METHOD TestTryWriteLRealMethod
VAR
    jsonParser : JsonDomParser;
    jsonInitialString : T_MAXSTRING := '{"foo":"bar"}';
    newLReal : LREAL := 12345.6789;  // Example LREAL value
    writeSuccess1 : BOOL;
    writeSuccess2 : BOOL;
    readLReal1 : LREAL;
    readLReal2 : LREAL;
    readResult1 : BOOL;
    readResult2 : BOOL;
    jsonOutput : T_MAXSTRING;
    expectedJsonOutput : T_MAXSTRING := '{"foo":"bar","myThing":[null,null,{"myLRealValue":12345.6789},null,12345.6789]}';
END_VAR
TEST('TestTryWriteLREALMethod');

// @TEST-RUN
jsonParser.ParseDocument(jsonInitialString);
writeSuccess1 := jsonParser.TryWrite('.myThing[2].myLRealValue', newLReal);
writeSuccess2 := jsonParser.TryWrite('.myThing[4]', newLReal);
jsonOutput := jsonParser.GetDocument();

readResult1 := jsonParser.TryRead('.myThing[2].myLRealValue', readLReal1);
readResult2 := jsonParser.TryRead('.myThing[4]', readLReal2);
jsonParser.NewDocument();

// @TEST-ASSERT
AssertTrue(Condition := writeSuccess1, Message := 'First TryWrite operation was unsuccessful for LREAL');
AssertTrue(Condition := writeSuccess2, Message := 'Second TryWrite operation was unsuccessful for LREAL');
AssertTrue(Condition := readResult1 AND ABS(readLReal1 - newLReal) < 1e-6, Message := 'Could not read back the first written LREAL value or value mismatched');  // using a tolerance for floating-point comparison
AssertTrue(Condition := readResult2 AND ABS(readLReal2 - newLReal) < 1e-6, Message := 'Could not read back the second written LREAL value or value mismatched');  // using a tolerance for floating-point comparison
AssertEquals(Expected := expectedJsonOutput, Actual := jsonOutput, Message := 'Output JSON does not match expected for LREAL');

TEST_FINISHED();
END_METHOD

METHOD TestTryWriteRealMethod
VAR
    jsonParser : JsonDomParser;
    jsonInitialString : T_MAXSTRING := '{"foo":"bar"}';
    newReal : REAL := 123.456;  // Example REAL value
    writeSuccess1 : BOOL;
    writeSuccess2 : BOOL;
    readReal1 : REAL;
    readReal2 : REAL;
    readResult1 : BOOL;
    readResult2 : BOOL;
    jsonOutput : T_MAXSTRING;
    expectedJsonOutput : T_MAXSTRING := '{"foo":"bar","myThing":[null,null,{"myRealValue":123.456},null,123.456]}';
END_VAR
TEST('TestTryWriteREALMethod');

// @TEST-RUN
jsonParser.ParseDocument(jsonInitialString);
writeSuccess1 := jsonParser.TryWrite('.myThing[2].myRealValue', newReal);
writeSuccess2 := jsonParser.TryWrite('.myThing[4]', newReal);
jsonOutput := jsonParser.GetDocument();

readResult1 := jsonParser.TryRead('.myThing[2].myRealValue', readReal1);
readResult2 := jsonParser.TryRead('.myThing[4]', readReal2);
jsonParser.NewDocument();

// @TEST-ASSERT
AssertTrue(Condition := writeSuccess1, Message := 'First TryWrite operation was unsuccessful for REAL');
AssertTrue(Condition := writeSuccess2, Message := 'Second TryWrite operation was unsuccessful for REAL');
AssertTrue(Condition := readResult1 AND ABS(readReal1 - newReal) < 1e-5, Message := 'Could not read back the first written REAL value or value mismatched');  // using a tolerance for floating-point comparison
AssertTrue(Condition := readResult2 AND ABS(readReal2 - newReal) < 1e-5, Message := 'Could not read back the second written REAL value or value mismatched');  // using a tolerance for floating-point comparison
//AssertEquals(Expected := expectedJsonOutput, Actual := jsonOutput, Message := 'Output JSON does not match expected for REAL');

TEST_FINISHED();
END_METHOD

METHOD TestTryWriteStringMethod
VAR
    jsonParser : JsonDomParser;
    jsonInitialString : T_MAXSTRING := '{"foo":"bar"}';
    newString : STRING := 'HelloWorld';  // Example STRING value
    writeSuccess1 : BOOL;
    writeSuccess2 : BOOL;
    readString1 : STRING;
    readString2 : STRING;
    readResult1 : BOOL;
    readResult2 : BOOL;
    jsonOutput : T_MAXSTRING;
    expectedJsonOutput : T_MAXSTRING := '{"foo":"bar","myThing":[null,null,{"myStringValue":"HelloWorld"},null,"HelloWorld"]}';
END_VAR
TEST('TestTryWriteSTRINGMethod');

// @TEST-RUN
jsonParser.ParseDocument(jsonInitialString);
writeSuccess1 := jsonParser.TryWrite('.myThing[2].myStringValue', newString);
writeSuccess2 := jsonParser.TryWrite('.myThing[4]', newString);
jsonOutput := jsonParser.GetDocument();

readResult1 := jsonParser.TryRead('.myThing[2].myStringValue', readString1);
readResult2 := jsonParser.TryRead('.myThing[4]', readString2);
jsonParser.NewDocument();

// @TEST-ASSERT
AssertTrue(Condition := writeSuccess1, Message := 'First TryWrite operation was unsuccessful for STRING');
AssertTrue(Condition := writeSuccess2, Message := 'Second TryWrite operation was unsuccessful for STRING');
AssertTrue(Condition := readResult1 AND (readString1 = newString), Message := 'Could not read back the first written STRING value or value mismatched');
AssertTrue(Condition := readResult2 AND (readString2 = newString), Message := 'Could not read back the second written STRING value or value mismatched');
AssertEquals(Expected := expectedJsonOutput, Actual := jsonOutput, Message := 'Output JSON does not match expected for STRING');

TEST_FINISHED();
END_METHOD

METHOD TestTryWriteUdintMethod
VAR
    jsonParser : JsonDomParser;
    jsonInitialString : T_MAXSTRING := '{"foo":"bar"}';
    newUDInt : UDINT := 1234567890;  // Assuming UDINT has a suitable range
    writeSuccess1 : BOOL;
    writeSuccess2 : BOOL;
    readUDInt1 : UDINT;
    readUDInt2 : UDINT;
    readResult1 : BOOL;
    readResult2 : BOOL;
    jsonOutput : T_MAXSTRING;
    expectedJsonOutput : T_MAXSTRING := '{"foo":"bar","myThing":[null,null,{"myUDIntValue":1234567890},null,1234567890]}';
END_VAR
TEST('TestTryWriteUDINTMethod');

// @TEST-RUN
jsonParser.ParseDocument(jsonInitialString);
writeSuccess1 := jsonParser.TryWrite('.myThing[2].myUDIntValue', newUDInt);
writeSuccess2 := jsonParser.TryWrite('.myThing[4]', newUDInt);
jsonOutput := jsonParser.GetDocument();

readResult1 := jsonParser.TryRead('.myThing[2].myUDIntValue', readUDInt1);
readResult2 := jsonParser.TryRead('.myThing[4]', readUDInt2);
jsonParser.NewDocument();

// @TEST-ASSERT
AssertTrue(Condition := writeSuccess1, Message := 'First TryWrite operation was unsuccessful for UDINT');
AssertTrue(Condition := writeSuccess2, Message := 'Second TryWrite operation was unsuccessful for UDINT');
AssertTrue(Condition := readResult1 AND (readUDInt1 = newUDInt), Message := 'Could not read back the first written UDINT value or value mismatched');
AssertTrue(Condition := readResult2 AND (readUDInt2 = newUDInt), Message := 'Could not read back the second written UDINT value or value mismatched');
AssertEquals(Expected := expectedJsonOutput, Actual := jsonOutput, Message := 'Output JSON does not match expected for UDINT');

TEST_FINISHED();
END_METHOD

END_FUNCTION_BLOCK

// ---- mobject-json/Tests/JsonSerializer_TestSuite.TcPOU
FUNCTION_BLOCK JsonSerializer_TestSuite EXTENDS TcUnit.FB_TestSuite

TestAddBase64();
TestAddBoolWithFalseBoolVariable();
TestAddBoolWithTrueBoolVariable();
TestAddByte();
TestAddBytesAsHex();
TestAddDateTime();
TestAddDcTime();
TestAddDint();
TestAddDword();
TestAddFileTime();
TestAddInt();
TestAddKey();
TestAddKeyBase64();
TestAddKeyBoolWithFalseBoolVariable();
TestAddKeyBoolWithTrueBoolVariable();
TestAddKeyByte();
TestAddKeyBytesAsHex();
TestAddKeyDateTime();
TestAddKeyDcTime();
TestAddKeyDint();
TestAddKeyDword();
TestAddKeyFileTime();
TestAddKeyInt();
TestAddKeyLint();
TestAddKeyLreal();
TestAddKeyLreal_Max();
TestAddKeyLtime();
TestAddKeyLword();
TestAddKeyNull();
TestAddKeyObject();
TestAddKeyObject_Array();
TestAddKeyRawJson();
TestAddKeyReal();
TestAddKeyReal_Max();
TestAddKeySint();
TestAddKeyString();
TestAddKeyStringByRef();
TestAddKeyTime();
TestAddKeyTod();
TestAddKeyUdint();
TestAddKeyUint();
TestAddKeyUlint();
TestAddKeyUsint();
TestAddKeyWord();
TestAddLint();
TestAddLreal();
TestAddLtime();
TestAddLword();
TestAddNull();
TestAddObject();
TestAddObjects();
TestAddRawJson();
TestAddReal();
TestAddSint();
TestAddString();
TestAddStringByRef();
TestAddTime();
TestAddTod();
TestAddUdint();
TestAddUint();
TestAddUlint();
TestAddUsint();
TestAddWord();
TestClone();
TestGetSerializedDataLengthEmpty();
TestGetSerializedDataLengthWithEmptyObject();
TestGetSerializedDataLengthWithSimpleObject();
TestReset();
TestSerializeArray();
TestSerializeObject();

METHOD PUBLIC TestAddBase64
VAR
	jsonSerializer : JsonSerializer;
	rawData : ARRAY[0..4] OF BYTE := [104, 101, 108, 108, 111];
	out : STRING;
	expected : STRING := '"aGVsbG8="';
END_VAR
TEST('TestAddBase64');

jsonSerializer.AddBase64(ADR(rawData), SIZEOF(rawData));
jsonSerializer.TryGetSerializedData(ADR(out),SIZEOF(out));

AssertEquals(
	Expected := expected,
	Actual := out,
	Message := 'Did not produce the expected JSON string for Base64 encoded "hello"'
);

TEST_FINISHED();
END_METHOD

METHOD PUBLIC TestAddBoolWithFalseBoolVariable
VAR
	jsonSerializer : JsonSerializer;
	value : BOOL := FALSE;
	out : STRING;
	expected : STRING := 'false';
END_VAR
TEST('TestAddBoolWithFalseBoolVariable');

jsonSerializer.AddBool(value);
jsonSerializer.TryGetSerializedData(ADR(out),SIZEOF(out));

AssertEquals(
	Expected := expected,
	Actual := out,
	Message := 'Did not produce the expected JSON string for a false value'
);

TEST_FINISHED();
END_METHOD

METHOD PUBLIC TestAddBoolWithTrueBoolVariable
VAR
	jsonSerializer : JsonSerializer;
	value : BOOL := TRUE;
	out : STRING;
	expected : STRING := 'true';
END_VAR
TEST('TestAddBoolWithTrueBoolVariable');

jsonSerializer.AddBool(value);
jsonSerializer.TryGetSerializedData(ADR(out),SIZEOF(out));

AssertEquals(
	Expected := expected,
	Actual := out,
	Message := 'Did not produce the expected JSON string for a true value'
);

TEST_FINISHED();
END_METHOD

METHOD PUBLIC TestAddByte
VAR
	jsonSerializer : JsonSerializer;
	byteValue : BYTE := 100;
	out : STRING;
	expected : STRING := '100';
END_VAR
TEST('TestAddByte');

jsonSerializer.AddByte(byteValue);
jsonSerializer.TryGetSerializedData(ADR(out),SIZEOF(out));

AssertEquals(
	Expected := expected,
	Actual := out,
	Message := 'Did not produce the expected JSON string for the BYTE value'
);

TEST_FINISHED();
END_METHOD

METHOD PUBLIC TestAddBytesAsHex
VAR
	jsonSerializer : JsonSerializer;
	binaryData : ARRAY[0..3] OF BYTE := [16#BA, 16#AD, 16#F0, 16#0D];
	out : STRING;
	expected : STRING := '"baadf00d"';
END_VAR
TEST('TestAddBytesAsHex');

jsonSerializer.AddBytesAsHex(ADR(binaryData), SIZEOF(binaryData));
jsonSerializer.TryGetSerializedData(ADR(out),SIZEOF(out));

AssertEquals(
	Expected := expected,
	Actual := out,
	Message := 'Did not produce the expected JSON string for hexadecimal binary data'
);

TEST_FINISHED();
END_METHOD

METHOD PUBLIC TestAddDateTime
VAR
	jsonSerializer : JsonSerializer;
	dateTimeValue : DATE_AND_TIME := DT#2023-12-30-15:20:00;
	out : STRING;
	expected : STRING := '"2023-12-30T15:20:00"';
END_VAR
TEST('TestAddDateTime');

jsonSerializer.AddDateTime(dateTimeValue);
jsonSerializer.TryGetSerializedData(ADR(out),SIZEOF(out));

AssertEquals(
	Expected := expected,
	Actual := out,
	Message := 'Did not produce the expected JSON string for the DATE_AND_TIME value'
);

TEST_FINISHED();
END_METHOD

METHOD PUBLIC TestAddDcTime
VAR
	jsonSerializer : JsonSerializer;
	dcTimeValue : DCTIME := 12345678;
	out : STRING;
	expected : STRING := '"2000-01-01T00:00:00.012345678"';
END_VAR
TEST('TestAddDcTime');

jsonSerializer.AddDcTime(dcTimeValue);
jsonSerializer.TryGetSerializedData(ADR(out),SIZEOF(out));

AssertEquals(
	Expected := expected,
	Actual := out,
	Message := 'Did not produce the expected JSON string for the DCTIME value'
);

TEST_FINISHED();
END_METHOD

METHOD PUBLIC TestAddDint
VAR
	jsonSerializer : JsonSerializer;
	dintValue : DINT := 12345;
	out : STRING;
	expected : STRING := '12345';
END_VAR
TEST('TestAddDint');

jsonSerializer.AddDint(dintValue);
jsonSerializer.TryGetSerializedData(ADR(out),SIZEOF(out));

AssertEquals(
	Expected := expected,
	Actual := out,
	Message := 'Did not produce the expected JSON string for the DINT value'
);

TEST_FINISHED();
END_METHOD

METHOD PUBLIC TestAddDword
VAR
	jsonSerializer : JsonSerializer;
	dwordValue : DWORD := 12345;
	out : STRING;
	expected : STRING := '12345';
END_VAR
TEST('TestAddDword');

jsonSerializer.AddDword(dwordValue);
jsonSerializer.TryGetSerializedData(ADR(out),SIZEOF(out));

AssertEquals(
	Expected := expected,
	Actual := out,
	Message := 'Did not produce the expected JSON string for the DWORD value'
);

TEST_FINISHED();
END_METHOD

METHOD PUBLIC TestAddFileTime
VAR
	jsonSerializer : JsonSerializer;
	fileTimeValue : FILETIME := 12345678;
	out : STRING;
	expected : STRING := '"1601-01-01T00:00:01.2345678"';
END_VAR
TEST('TestAddFileTime');

jsonSerializer.AddFileTime(fileTimeValue);
jsonSerializer.TryGetSerializedData(ADR(out),SIZEOF(out));

AssertEquals(
	Expected := expected,
	Actual := out,
	Message := 'Did not produce the expected JSON string for the FileTime value'
);

TEST_FINISHED();
END_METHOD

METHOD PUBLIC TestAddInt
VAR
	jsonSerializer : JsonSerializer;
	intValue : INT := 12345;
	out : STRING;
	expected : STRING := '12345';
END_VAR
TEST('TestAddInt');

jsonSerializer.AddInt(intValue);
jsonSerializer.TryGetSerializedData(ADR(out),SIZEOF(out));

AssertEquals(
	Expected := expected,
	Actual := out,
	Message := 'Did not produce the expected JSON string for the INT value'
);

TEST_FINISHED();
END_METHOD

METHOD PUBLIC TestAddKey
VAR
	jsonSerializer : JsonSerializer;
	out : STRING;
	expected : STRING := '{"data":123}';
END_VAR
TEST('TestAddKey');

jsonSerializer.StartObject();
jsonSerializer.AddKey('data');
jsonSerializer.AddDint(123);
jsonSerializer.EndObject();

jsonSerializer.TryGetSerializedData(ADR(out),SIZEOF(out));

AssertEquals(
	Expected := expected,
	Actual := out,
	Message := 'Did not produce the expected JSON string for the KEY value'
);

TEST_FINISHED();
END_METHOD

METHOD PUBLIC TestAddKeyBase64
VAR
	jsonSerializer : JsonSerializer;
	rawData : ARRAY[0..4] OF BYTE := [104, 101, 108, 108, 111];
	out : STRING;
	expected : STRING := '{"data":"aGVsbG8="}';
END_VAR
TEST('TestAddKeyBase64');

jsonSerializer.StartObject();
jsonSerializer.AddKeyBase64('data',ADR(rawData), SIZEOF(rawData));
jsonSerializer.EndObject();

jsonSerializer.TryGetSerializedData(ADR(out),SIZEOF(out));

AssertEquals(
	Expected := expected,
	Actual := out,
	Message := 'Did not produce the expected JSON string for Base64 encoded "hello"'
);

TEST_FINISHED();
END_METHOD

METHOD PUBLIC TestAddKeyBoolWithFalseBoolVariable
VAR
	jsonSerializer : JsonSerializer;
	value : BOOL := FALSE;
	out : STRING;
	expected : STRING := '{"data":false}';
END_VAR
TEST('TestAddKeyBoolWithFalseBoolVariable');

jsonSerializer.StartObject();
jsonSerializer.AddKeyBool('data',value);
jsonSerializer.EndObject();

jsonSerializer.TryGetSerializedData(ADR(out),SIZEOF(out));

AssertEquals(
	Expected := expected,
	Actual := out,
	Message := 'Did not produce the expected JSON string for a false value'
);

TEST_FINISHED();
END_METHOD

METHOD PUBLIC TestAddKeyBoolWithTrueBoolVariable
VAR
	jsonSerializer : JsonSerializer;
	value : BOOL := TRUE;
	out : STRING;
	expected : STRING := '{"data":true}';
END_VAR
TEST('TestAddKeyBoolWithTrueBoolVariable');

jsonSerializer.StartObject();
jsonSerializer.AddKeyBool('data',value);
jsonSerializer.EndObject();

jsonSerializer.TryGetSerializedData(ADR(out),SIZEOF(out));

AssertEquals(
	Expected := expected,
	Actual := out,
	Message := 'Did not produce the expected JSON string for a true value'
);

TEST_FINISHED();
END_METHOD

METHOD PUBLIC TestAddKeyByte
VAR
	jsonSerializer : JsonSerializer;
	byteValue : BYTE := 100;
	out : STRING;
	expected : STRING := '{"data":100}';
END_VAR
TEST('TestAddKeyByte');

jsonSerializer.StartObject();
jsonSerializer.AddKeyByte('data',byteValue);
jsonSerializer.EndObject();

jsonSerializer.TryGetSerializedData(ADR(out),SIZEOF(out));

AssertEquals(
	Expected := expected,
	Actual := out,
	Message := 'Did not produce the expected JSON string for the BYTE value'
);

TEST_FINISHED();
END_METHOD

METHOD PUBLIC TestAddKeyBytesAsHex
VAR
	jsonSerializer : JsonSerializer;
	binaryData : ARRAY[0..3] OF BYTE := [16#BA, 16#AD, 16#F0, 16#0D];
	out : STRING;
	expected : STRING := '{"data":"baadf00d"}';
END_VAR
TEST('TestAddKeyBytesAsHex');

jsonSerializer.StartObject();
jsonSerializer.AddKeyBytesAsHex('data',ADR(binaryData), SIZEOF(binaryData));
jsonSerializer.EndObject();

jsonSerializer.TryGetSerializedData(ADR(out),SIZEOF(out));

AssertEquals(
	Expected := expected,
	Actual := out,
	Message := 'Did not produce the expected JSON string for hexadecimal binary data'
);

TEST_FINISHED();
END_METHOD

METHOD PUBLIC TestAddKeyDateTime
VAR
	jsonSerializer : JsonSerializer;
	dateTimeValue : DATE_AND_TIME := DT#2023-12-30-15:20:00;
	out : STRING;
	expected : STRING := '{"data":"2023-12-30T15:20:00"}';
END_VAR
TEST('TestAddKeyDateTime');

jsonSerializer.StartObject();
jsonSerializer.AddKeyDateTime('data',dateTimeValue);
jsonSerializer.EndObject();

jsonSerializer.TryGetSerializedData(ADR(out),SIZEOF(out));

AssertEquals(
	Expected := expected,
	Actual := out,
	Message := 'Did not produce the expected JSON string for the DATE_AND_TIME value'
);

TEST_FINISHED();
END_METHOD

METHOD PUBLIC TestAddKeyDcTime
VAR
	jsonSerializer : JsonSerializer;
	dcTimeValue : DCTIME := 12345678;
	out : STRING;
	expected : STRING := '{"data":"2000-01-01T00:00:00.012345678"}';
END_VAR
TEST('TestAddKeyDcTime');

jsonSerializer.StartObject();
jsonSerializer.AddKeyDcTime('data',dcTimeValue);
jsonSerializer.EndObject();

jsonSerializer.TryGetSerializedData(ADR(out),SIZEOF(out));

AssertEquals(
	Expected := expected,
	Actual := out,
	Message := 'Did not produce the expected JSON string for the DCTIME value'
);

TEST_FINISHED();
END_METHOD

METHOD PUBLIC TestAddKeyDint
VAR
	jsonSerializer : JsonSerializer;
	dintValue : DINT := 12345;
	out : STRING;
	expected : STRING := '{"data":12345}';
END_VAR
TEST('TestAddKeyDint');

jsonSerializer.StartObject();
jsonSerializer.AddKeyDint('data',dintValue);
jsonSerializer.EndObject();

jsonSerializer.TryGetSerializedData(ADR(out),SIZEOF(out));

AssertEquals(
	Expected := expected,
	Actual := out,
	Message := 'Did not produce the expected JSON string for the DINT value'
);

TEST_FINISHED();
END_METHOD

METHOD PUBLIC TestAddKeyDword
VAR
	jsonSerializer : JsonSerializer;
	dwordValue : DWORD := 12345;
	out : STRING;
	expected : STRING := '{"data":12345}';
END_VAR
TEST('TestAddKeyDword');

jsonSerializer.StartObject();
jsonSerializer.AddKeyDword('data',dwordValue);
jsonSerializer.EndObject();

jsonSerializer.TryGetSerializedData(ADR(out),SIZEOF(out));

AssertEquals(
	Expected := expected,
	Actual := out,
	Message := 'Did not produce the expected JSON string for the DWORD value'
);

TEST_FINISHED();
END_METHOD

METHOD PUBLIC TestAddKeyFileTime
VAR
	jsonSerializer : JsonSerializer;
	fileTimeValue : FILETIME := 12345678;
	out : STRING;
	expected : STRING := '{"data":"1601-01-01T00:00:01.2345678"}';
END_VAR
TEST('TestAddKeyFileTime');

jsonSerializer.StartObject();
jsonSerializer.AddKeyFileTime('data',fileTimeValue);
jsonSerializer.EndObject();

jsonSerializer.TryGetSerializedData(ADR(out),SIZEOF(out));

AssertEquals(
	Expected := expected,
	Actual := out,
	Message := 'Did not produce the expected JSON string for the FileTime value'
);

TEST_FINISHED();
END_METHOD

METHOD PUBLIC TestAddKeyInt
VAR
	jsonSerializer : JsonSerializer;
	intValue : INT := 12345;
	out : STRING;
	expected : STRING := '{"data":12345}';
END_VAR
TEST('TestAddKeyInt');

jsonSerializer.StartObject();
jsonSerializer.AddKeyInt('data',intValue);
jsonSerializer.EndObject();

jsonSerializer.TryGetSerializedData(ADR(out),SIZEOF(out));

AssertEquals(
	Expected := expected,
	Actual := out,
	Message := 'Did not produce the expected JSON string for the INT value'
);

TEST_FINISHED();
END_METHOD

METHOD PUBLIC TestAddKeyLint
VAR
	jsonSerializer : JsonSerializer;
	lintValue : LINT := 9223372036854775807;
	out : STRING;
	expected : STRING := '{"data":9223372036854775807}';
END_VAR
TEST('TestAddKeyLint');

jsonSerializer.StartObject();
jsonSerializer.AddKeyLint('data',lintValue);
jsonSerializer.EndObject();

jsonSerializer.TryGetSerializedData(ADR(out),SIZEOF(out));

AssertEquals(
	Expected := expected,
	Actual := out,
	Message := 'Did not produce the expected JSON string for the LINT value'
);

TEST_FINISHED();
END_METHOD

METHOD PUBLIC TestAddKeyLreal
VAR
	jsonSerializer : JsonSerializer;
	lrealValue : LREAL := 123456.789;
	out : STRING;
	expected : STRING := '{"data":123456.789}';
END_VAR
TEST('TestAddKeyLreal');

jsonSerializer.StartObject();
jsonSerializer.AddKeyLreal('data',lrealValue);
jsonSerializer.EndObject();

jsonSerializer.TryGetSerializedData(ADR(out),SIZEOF(out));

AssertEquals(
	Expected := expected,
	Actual := out,
	Message := 'Did not produce the expected JSON string for the LREAL value'
);

TEST_FINISHED();
END_METHOD

METHOD PUBLIC TestAddKeyLreal_Max
VAR
	jsonSerializer : JsonSerializer;
	lrealValue : LREAL := DatatypeLimits.LREAL_MAX_VALUE;
	out : STRING;
	expected : STRING := '{"data":1.7976931348623157e308}';
END_VAR
TEST('TestAddKeyLreal_Max');

jsonSerializer.StartObject();
jsonSerializer.AddKeyLreal('data',lrealValue);
jsonSerializer.EndObject();

jsonSerializer.TryGetSerializedData(ADR(out),SIZEOF(out));

AssertEquals(
	Expected := expected,
	Actual := out,
	Message := 'Did not produce the expected JSON string for the LREAL value'
);

TEST_FINISHED();
END_METHOD

METHOD PUBLIC TestAddKeyLtime
VAR
	jsonSerializer : JsonSerializer;
	ltimeValue : LTIME := LTIME#100D2H30M40S500MS600US700NS;
	out : STRING;
	expected : STRING := '{"data":"LTIME#100d2h30m40s500ms600us700ns"}';
END_VAR
TEST('TestAddKeyLtime');

jsonSerializer.StartObject();
jsonSerializer.AddKeyLtime('data',ltimeValue);
jsonSerializer.EndObject();

jsonSerializer.TryGetSerializedData(ADR(out),SIZEOF(out));

AssertEquals(
	Expected := expected,
	Actual := out,
	Message := 'Did not produce the expected JSON string for the LTIME value'
);

TEST_FINISHED();
END_METHOD

METHOD PUBLIC TestAddKeyLword
VAR
	jsonSerializer : JsonSerializer;
	lwordValue : LWORD := 9223372036854775807;
	out : STRING;
	expected : STRING := '{"data":9223372036854775807}';
END_VAR
TEST('TestAddKeyLword');

jsonSerializer.StartObject();
jsonSerializer.AddKeyLword('data',lwordValue);
jsonSerializer.EndObject();

jsonSerializer.TryGetSerializedData(ADR(out),SIZEOF(out));

AssertEquals(
	Expected := expected,
	Actual := out,
	Message := 'Did not produce the expected JSON string for the LWORD value'
);

TEST_FINISHED();
END_METHOD

METHOD PUBLIC TestAddKeyNull
VAR
	jsonSerializer : JsonSerializer;
	out : STRING;
	expected : STRING := '{"data":null}';
END_VAR
TEST('TestAddKeyNull');

jsonSerializer.StartObject();
jsonSerializer.AddKeyNull('data');
jsonSerializer.EndObject();

jsonSerializer.TryGetSerializedData(ADR(out),SIZEOF(out));

AssertEquals(
	Expected := expected,
	Actual := out,
	Message := 'Did not produce the expected JSON string for the NULL value'
);

TEST_FINISHED();
END_METHOD

METHOD PUBLIC TestAddKeyObject
VAR
	jsonSerializer : JsonSerializer;
	user : MockSerializableUserObject(Name := 'alice', Age := 40);
	out : STRING;
	expected : STRING := '{"data":{"Name":"alice","Age":40}}';
END_VAR
TEST('TestAddKeyObject');

jsonSerializer.StartObject();
jsonSerializer.AddKeyObject('data',user);
jsonSerializer.EndObject();

jsonSerializer.TryGetSerializedData(ADR(out),SIZEOF(out));

AssertEquals(
	Expected := expected,
	Actual := out,
	Message := 'Did not produce the expected JSON string for the Object value'
);

TEST_FINISHED();
END_METHOD

METHOD PUBLIC TestAddKeyObject_Array
VAR
	jsonSerializer : JsonSerializer;
	user : MockSerializableArray(Name := 'alice', Age := 40);
	out : STRING;
	expected : STRING := '{"data":["alice",40]}';
END_VAR
TEST('TestAddKeyObject_Array');

jsonSerializer.StartObject();
jsonSerializer.AddKeyObject('data',user);
jsonSerializer.EndObject();

jsonSerializer.TryGetSerializedData(ADR(out),SIZEOF(out));

AssertEquals(
	Expected := expected,
	Actual := out,
	Message := 'Did not produce the expected JSON string for the Object value'
);

TEST_FINISHED();
END_METHOD

METHOD PUBLIC TestAddKeyRawJson
VAR
	jsonSerializer : JsonSerializer;
	rawObject : STRING := '{"foo":"bar"}';
	out : STRING;
	expected : STRING := '{"data":{"foo":"bar"}}';
END_VAR
TEST('TestAddKeyRawJson');

jsonSerializer.StartObject();
jsonSerializer.AddKeyRawJson('data',rawObject);
jsonSerializer.EndObject();

jsonSerializer.TryGetSerializedData(ADR(out),SIZEOF(out));

AssertEquals(
	Expected := expected,
	Actual := out,
	Message := 'Did not produce the expected JSON string for the raw object value'
);

TEST_FINISHED();
END_METHOD

METHOD PUBLIC TestAddKeyReal
VAR
	jsonSerializer : JsonSerializer;
	realValue : REAL := 123.4;
	out : STRING;
	expected : STRING := '{"data":123.4000015258789}'; // this has been adapted to support more decimal places, due to the issue with REAL conversion in TwinCAT 4024.56
END_VAR
TEST('TestAddKeyReal');

jsonSerializer.StartObject();
jsonSerializer.AddKeyReal('data',realValue);
jsonSerializer.EndObject();

jsonSerializer.TryGetSerializedData(ADR(out),SIZEOF(out));

AssertEquals(
	Expected := expected,
	Actual := out,
	Message := 'Did not produce the expected JSON string for the REAL value'
);

TEST_FINISHED();
END_METHOD

METHOD PUBLIC TestAddKeyReal_Max
VAR
	jsonSerializer : JsonSerializer;
	realValue : REAL := DatatypeLimits.REAL_MAX_VALUE;
	out : STRING;
	expected : STRING := '{"data":3.4028230607370965e38}'; // this has been adapted to support more decimal places, due to the issue with REAL conversion in TwinCAT 4024.56
END_VAR
TEST('TestAddKeyReal_Max');

jsonSerializer.StartObject();
jsonSerializer.AddKeyReal('data',realValue);
jsonSerializer.EndObject();

jsonSerializer.TryGetSerializedData(ADR(out),SIZEOF(out));

AssertEquals(
	Expected := expected,
	Actual := out,
	Message := 'Did not produce the expected JSON string for the REAL value'
);

TEST_FINISHED();
END_METHOD

METHOD PUBLIC TestAddKeySint
VAR
	jsonSerializer : JsonSerializer;
	sintValue : SINT := 123;
	out : STRING;
	expected : STRING := '{"data":123}';
END_VAR
TEST('TestAddKeySint');

jsonSerializer.StartObject();
jsonSerializer.AddKeySint('data',sintValue);
jsonSerializer.EndObject();

jsonSerializer.TryGetSerializedData(ADR(out),SIZEOF(out));

AssertEquals(
	Expected := expected,
	Actual := out,
	Message := 'Did not produce the expected JSON string for the SINT value'
);

TEST_FINISHED();
END_METHOD

METHOD PUBLIC TestAddKeyString
VAR
	jsonSerializer : JsonSerializer;
	stringValue : STRING := 'foobar';
	out : STRING;
	expected : STRING := '{"data":"foobar"}';
END_VAR
TEST('TestAddKeyString');

jsonSerializer.StartObject();
jsonSerializer.AddKeyString('data',stringValue);
jsonSerializer.EndObject();

jsonSerializer.TryGetSerializedData(ADR(out),SIZEOF(out));

AssertEquals(
	Expected := expected,
	Actual := out,
	Message := 'Did not produce the expected JSON string for the STRING value'
);

TEST_FINISHED();
END_METHOD

METHOD PUBLIC TestAddKeyStringByRef
VAR
	jsonSerializer : JsonSerializer;
	stringValue : T_MAXSTRING := '1234567890123456789012345678901234567890123456789012345678901234567890123456789012345678901234567890';
	out : T_MAXSTRING;
	expected : T_MAXSTRING := '{"data":"1234567890123456789012345678901234567890123456789012345678901234567890123456789012345678901234567890"}';
END_VAR
TEST('TestAddKeyStringByRef');

jsonSerializer.StartObject();
jsonSerializer.AddKeyStringByRef('data',stringValue);
jsonSerializer.EndObject();

jsonSerializer.TryGetSerializedData(ADR(out),SIZEOF(out));

AssertEquals(
	Expected := expected,
	Actual := out,
	Message := 'Did not produce the expected JSON string for the STRING using reference value'
);

TEST_FINISHED();
END_METHOD

METHOD PUBLIC TestAddKeyTime
VAR
	jsonSerializer : JsonSerializer;
	timeValue : TIME := T#49D17H2M47S295MS;
	out : STRING;
	expected : STRING := '{"data":"T#49d17h2m47s295ms"}';
END_VAR
TEST('TestAddKeyTime');

jsonSerializer.StartObject();
jsonSerializer.AddKeyTime('data',timeValue);
jsonSerializer.EndObject();

jsonSerializer.TryGetSerializedData(ADR(out),SIZEOF(out));

AssertEquals(
	Expected := expected,
	Actual := out,
	Message := 'Did not produce the expected JSON string for the TIME value'
);

TEST_FINISHED();
END_METHOD

METHOD PUBLIC TestAddKeyTod
VAR
	jsonSerializer : JsonSerializer;
	todValue : TOD := TOD#23:01:23.456;
	out : STRING;
	expected : STRING := '{"data":"TOD#23:01:23.456"}';
END_VAR
TEST('TestAddKeyTod');

jsonSerializer.StartObject();
jsonSerializer.AddKeyTod('data',todValue);
jsonSerializer.EndObject();

jsonSerializer.TryGetSerializedData(ADR(out),SIZEOF(out));

AssertEquals(
	Expected := expected,
	Actual := out,
	Message := 'Did not produce the expected JSON string for the TOD value'
);

TEST_FINISHED();
END_METHOD

METHOD PUBLIC TestAddKeyUdint
VAR
	jsonSerializer : JsonSerializer;
	udintValue : UDINT := 123456;
	out : STRING;
	expected : STRING := '{"data":123456}';
END_VAR
TEST('TestAddKeyUdint');

jsonSerializer.StartObject();
jsonSerializer.AddKeyUdint('data',udintValue);
jsonSerializer.EndObject();

jsonSerializer.TryGetSerializedData(ADR(out),SIZEOF(out));

AssertEquals(
	Expected := expected,
	Actual := out,
	Message := 'Did not produce the expected JSON string for the UDINT value'
);

TEST_FINISHED();
END_METHOD

METHOD PUBLIC TestAddKeyUint
VAR
	jsonSerializer : JsonSerializer;
	uintValue : UINT := 12345;
	out : STRING;
	expected : STRING := '{"data":12345}';
END_VAR
TEST('TestAddKeyUint');

jsonSerializer.StartObject();
jsonSerializer.AddKeyUint('data',uintValue);
jsonSerializer.EndObject();

jsonSerializer.TryGetSerializedData(ADR(out),SIZEOF(out));

AssertEquals(
	Expected := expected,
	Actual := out,
	Message := 'Did not produce the expected JSON string for the UINT value'
);

TEST_FINISHED();
END_METHOD

METHOD PUBLIC TestAddKeyUlint
VAR
	jsonSerializer : JsonSerializer;
	ulintValue : ULINT := 9223372036854775807;
	out : STRING;
	expected : STRING := '{"data":9223372036854775807}';
END_VAR
TEST('TestAddKeyUlint');

jsonSerializer.StartObject();
jsonSerializer.AddKeyUlint('data',ulintValue);
jsonSerializer.EndObject();

jsonSerializer.TryGetSerializedData(ADR(out),SIZEOF(out));

AssertEquals(
	Expected := expected,
	Actual := out,
	Message := 'Did not produce the expected JSON string for the ULINT value'
);

TEST_FINISHED();
END_METHOD

METHOD PUBLIC TestAddKeyUsint
VAR
	jsonSerializer : JsonSerializer;
	usintValue : USINT := 123;
	out : STRING;
	expected : STRING := '{"data":123}';
END_VAR
TEST('TestAddKeyUsint');

jsonSerializer.StartObject();
jsonSerializer.AddKeyUsint('data',usintValue);
jsonSerializer.EndObject();

jsonSerializer.TryGetSerializedData(ADR(out),SIZEOF(out));

AssertEquals(
	Expected := expected,
	Actual := out,
	Message := 'Did not produce the expected JSON string for the USINT value'
);

TEST_FINISHED();
END_METHOD

METHOD PUBLIC TestAddKeyWord
VAR
	jsonSerializer : JsonSerializer;
	wordValue : WORD := 12345;
	out : STRING;
	expected : STRING := '{"data":12345}';
END_VAR
TEST('TestAddKeyWord');

jsonSerializer.StartObject();
jsonSerializer.AddKeyWord('data',wordValue);
jsonSerializer.EndObject();

jsonSerializer.TryGetSerializedData(ADR(out),SIZEOF(out));

AssertEquals(
	Expected := expected,
	Actual := out,
	Message := 'Did not produce the expected JSON string for the WORD value'
);

TEST_FINISHED();
END_METHOD

METHOD PUBLIC TestAddLint
VAR
	jsonSerializer : JsonSerializer;
	lintValue : LINT := 9223372036854775807;
	out : STRING;
	expected : STRING := '9223372036854775807';
END_VAR
TEST('TestAddLint');

jsonSerializer.AddLint(lintValue);
jsonSerializer.TryGetSerializedData(ADR(out),SIZEOF(out));

AssertEquals(
	Expected := expected,
	Actual := out,
	Message := 'Did not produce the expected JSON string for the LINT value'
);

TEST_FINISHED();
END_METHOD

METHOD PUBLIC TestAddLreal
VAR
	jsonSerializer : JsonSerializer;
	lrealValue : LREAL := 123456.789;
	out : STRING;
	expected : STRING := '123456.789';
END_VAR
TEST('TestAddLReal');

jsonSerializer.AddLreal(lrealValue);
jsonSerializer.TryGetSerializedData(ADR(out),SIZEOF(out));

AssertEquals(
	Expected := expected,
	Actual := out,
	Message := 'Did not produce the expected JSON string for the LREAL value'
);

TEST_FINISHED();
END_METHOD

METHOD PUBLIC TestAddLtime
VAR
	jsonSerializer : JsonSerializer;
	ltimeValue : LTIME := LTIME#100D2H30M40S500MS600US700NS;
	out : STRING;
	expected : STRING := '"LTIME#100d2h30m40s500ms600us700ns"';
END_VAR
TEST('TestAddLtime');

jsonSerializer.AddLtime(ltimeValue);
jsonSerializer.TryGetSerializedData(ADR(out),SIZEOF(out));

AssertEquals(
	Expected := expected,
	Actual := out,
	Message := 'Did not produce the expected JSON string for the LTIME value'
);

TEST_FINISHED();
END_METHOD

METHOD PUBLIC TestAddLword
VAR
	jsonSerializer : JsonSerializer;
	lwordValue : LWORD := 9223372036854775807;
	out : STRING;
	expected : STRING := '9223372036854775807';
END_VAR
TEST('TestAddLword');

jsonSerializer.AddLword(lwordValue);
jsonSerializer.TryGetSerializedData(ADR(out),SIZEOF(out));

AssertEquals(
	Expected := expected,
	Actual := out,
	Message := 'Did not produce the expected JSON string for the LWORD value'
);

TEST_FINISHED();
END_METHOD

METHOD PUBLIC TestAddNull
VAR
	jsonSerializer : JsonSerializer;
	out : STRING;
	expected : STRING := 'null';
END_VAR
TEST('TestAddNull');

jsonSerializer.AddNull();
jsonSerializer.TryGetSerializedData(ADR(out),SIZEOF(out));

AssertEquals(
	Expected := expected,
	Actual := out,
	Message := 'Did not produce the expected JSON string for the NULL value'
);

TEST_FINISHED();
END_METHOD

METHOD PUBLIC TestAddObject
VAR
	jsonSerializer : JsonSerializer;
	user : MockSerializableUserObject(Name := 'alice', Age := 40);
	out : STRING;
	expected : STRING := '{"Name":"alice","Age":40}';
END_VAR
TEST('TestAddObject');

jsonSerializer.AddObject(user);
jsonSerializer.TryGetSerializedData(ADR(out),SIZEOF(out));

AssertEquals(
	Expected := expected,
	Actual := out,
	Message := 'Did not produce the expected JSON string for the Object value'
);

TEST_FINISHED();
END_METHOD

METHOD PUBLIC TestAddObjects
VAR
	jsonSerializer : JsonSerializer;
	user1 : MockSerializableUserObject(Name := 'alice', Age := 40);
    user2 : MockSerializableUserObject(Name := 'bob', Age := 50);
	out : STRING;
	expected : STRING := '{"users":[{"Name":"alice","Age":40},{"Name":"bob","Age":50}]}';
END_VAR
TEST('TestAddObjects');

jsonSerializer.StartObject();
jsonSerializer.AddKey('users');
jsonSerializer.StartArray();
jsonSerializer.AddObject(user1);
jsonSerializer.AddObject(user2);
jsonSerializer.EndArray();
jsonSerializer.EndObject();
jsonSerializer.TryGetSerializedData(ADR(out),SIZEOF(out));

AssertEquals(
	Expected := expected,
	Actual := out,
	Message := 'Did not produce the expected JSON string for the Object value'
);

TEST_FINISHED();
END_METHOD

METHOD PUBLIC TestAddRawJson
VAR
	jsonSerializer : JsonSerializer;
	rawObject : STRING := '{"foo":"bar"}';
	out : STRING;
	expected : STRING := '{"foo":"bar"}';
END_VAR
TEST('TestAddRawJson');

jsonSerializer.AddRawJson(rawObject);
jsonSerializer.TryGetSerializedData(ADR(out),SIZEOF(out));

AssertEquals(
	Expected := expected,
	Actual := out,
	Message := 'Did not produce the expected JSON string for the raw object value'
);

TEST_FINISHED();
END_METHOD

METHOD PUBLIC TestAddReal
VAR
	jsonSerializer : JsonSerializer;
	realValue : REAL := 123.4;
	out : STRING;
	expected : STRING := '123.4000015258789'; // this has been adapted to support more decimal places, due to the issue with REAL conversion in TwinCAT 4024.56
END_VAR
TEST('TestAddReal');

jsonSerializer.AddReal(realValue);
jsonSerializer.TryGetSerializedData(ADR(out),SIZEOF(out));

AssertEquals(
	Expected := expected,
	Actual := out,
	Message := 'Did not produce the expected JSON string for the REAL value'
);

TEST_FINISHED();
END_METHOD

METHOD PUBLIC TestAddSint
VAR
	jsonSerializer : JsonSerializer;
	intValue : SINT := 123;
	out : STRING;
	expected : STRING := '123';
END_VAR
TEST('TestAddSint');

jsonSerializer.AddSint(intValue);
jsonSerializer.TryGetSerializedData(ADR(out),SIZEOF(out));

AssertEquals(
	Expected := expected,
	Actual := out,
	Message := 'Did not produce the expected JSON string for the SINT value'
);

TEST_FINISHED();
END_METHOD

METHOD PUBLIC TestAddString
VAR
	jsonSerializer : JsonSerializer;
	stringValue : STRING := 'foobar';
	out : STRING;
	expected : STRING := '"foobar"';
END_VAR
TEST('TestAddString');

jsonSerializer.AddString(stringValue);
jsonSerializer.TryGetSerializedData(ADR(out),SIZEOF(out));

AssertEquals(
	Expected := expected,
	Actual := out,
	Message := 'Did not produce the expected JSON string for the STRING value'
);

TEST_FINISHED();
END_METHOD

METHOD PUBLIC TestAddStringByRef
VAR
	jsonSerializer : JsonSerializer;
	stringValue : T_MAXSTRING := '1234567890123456789012345678901234567890123456789012345678901234567890123456789012345678901234567890';
	out : T_MAXSTRING;
	expected : T_MAXSTRING := '"1234567890123456789012345678901234567890123456789012345678901234567890123456789012345678901234567890"';
END_VAR
TEST('TestAddStringByRef');

jsonSerializer.AddStringByRef(stringValue);
jsonSerializer.TryGetSerializedData(ADR(out),SIZEOF(out));

AssertEquals(
	Expected := expected,
	Actual := out,
	Message := 'Did not produce the expected JSON string for the STRING using reference value'
);

TEST_FINISHED();
END_METHOD

METHOD PUBLIC TestAddTime
VAR
	jsonSerializer : JsonSerializer;
	timeValue : TIME := T#49D17H2M47S295MS;
	out : STRING;
	expected : STRING := '"T#49d17h2m47s295ms"';
END_VAR
TEST('TestAddTime');

jsonSerializer.AddTime(timeValue);
jsonSerializer.TryGetSerializedData(ADR(out),SIZEOF(out));

AssertEquals(
	Expected := expected,
	Actual := out,
	Message := 'Did not produce the expected JSON string for the TIME value'
);

TEST_FINISHED();
END_METHOD

METHOD PUBLIC TestAddTod
VAR
	jsonSerializer : JsonSerializer;
	todValue : TOD := TOD#23:01:23.456;
	out : STRING;
	expected : STRING := '"TOD#23:01:23.456"';
END_VAR
TEST('TestAddTod');

jsonSerializer.AddTod(todValue);
jsonSerializer.TryGetSerializedData(ADR(out),SIZEOF(out));

AssertEquals(
	Expected := expected,
	Actual := out,
	Message := 'Did not produce the expected JSON string for the TOD value'
);

TEST_FINISHED();
END_METHOD

METHOD PUBLIC TestAddUdint
VAR
	jsonSerializer : JsonSerializer;
	udintValue : UDINT := 123456;
	out : STRING;
	expected : STRING := '123456';
END_VAR
TEST('TestAddUdint');

jsonSerializer.AddUdint(udintValue);
jsonSerializer.TryGetSerializedData(ADR(out),SIZEOF(out));

AssertEquals(
	Expected := expected,
	Actual := out,
	Message := 'Did not produce the expected JSON string for the UDINT value'
);

TEST_FINISHED();
END_METHOD

METHOD PUBLIC TestAddUint
VAR
	jsonSerializer : JsonSerializer;
	uintValue : UINT := 12345;
	out : STRING;
	expected : STRING := '12345';
END_VAR
TEST('TestAddUint');


jsonSerializer.AddUint(uintValue);
jsonSerializer.TryGetSerializedData(ADR(out),SIZEOF(out));

AssertEquals(
	Expected := expected,
	Actual := out,
	Message := 'Did not produce the expected JSON string for the UINT value'
);

TEST_FINISHED();
END_METHOD

METHOD PUBLIC TestAddUlint
VAR
	jsonSerializer : JsonSerializer;
	ulintValue : ULINT := 9223372036854775807;
	out : STRING;
	expected : STRING := '9223372036854775807';
END_VAR
TEST('TestAddUlint');

jsonSerializer.AddUlint(ulintValue);
jsonSerializer.TryGetSerializedData(ADR(out),SIZEOF(out));

AssertEquals(
	Expected := expected,
	Actual := out,
	Message := 'Did not produce the expected JSON string for the ULINT value'
);

TEST_FINISHED();
END_METHOD

METHOD PUBLIC TestAddUsint
VAR
	jsonSerializer : JsonSerializer;
	usintValue : USINT := 123;
	out : STRING;
	expected : STRING := '123';
END_VAR
TEST('TestAddUsint');

jsonSerializer.AddUsint(usintValue);
jsonSerializer.TryGetSerializedData(ADR(out),SIZEOF(out));

AssertEquals(
	Expected := expected,
	Actual := out,
	Message := 'Did not produce the expected JSON string for the USINT value'
);

TEST_FINISHED();
END_METHOD

METHOD PUBLIC TestAddWord
VAR
	jsonSerializer : JsonSerializer;
	wordValue : WORD := 12345;
	out : STRING;
	expected : STRING := '12345';
END_VAR
TEST('TestAddWord');

jsonSerializer.AddWord(wordValue);
jsonSerializer.TryGetSerializedData(ADR(out),SIZEOF(out));

AssertEquals(
	Expected := expected,
	Actual := out,
	Message := 'Did not produce the expected JSON string for the WORD value'
);

TEST_FINISHED();
END_METHOD

METHOD PUBLIC TestClone
VAR
	jsonSerializer : JsonSerializer;
	clone : I_Serializer;
	rawObject : STRING := '{"foo":"bar"}';
	out : STRING;
	expected : STRING := '{"foo":"bar"}';
END_VAR
TEST('TestClone');

// add something to the original 
jsonSerializer.AddRawJson(rawObject);

// deep clone
clone := jsonSerializer.Clone();

// reset the original
jsonSerializer.Reset();

// retreive the data from the clone
clone.TryGetSerializedData(ADR(out),SIZEOF(out));

// clones are __NEW so must be disposed
clone.Dispose();

AssertEquals(
	Expected := expected,
	Actual := out,
	Message := 'Did not create a deep copy clone'
);

TEST_FINISHED();
END_METHOD

METHOD PUBLIC TestGetSerializedDataLengthEmpty
VAR
	jsonSerializer : JsonSerializer;
	rawObject : STRING := '';
	length : UDINT;
	expected : UDINT := 0;
END_VAR
TEST('TestGetSerializedDataLengthEmpty');

length := jsonSerializer.GetSerializedDataLength();

AssertEquals(
	Expected := expected,
	Actual := length,
	Message := 'Did not produce the expected JSON string length'
);

TEST_FINISHED();
END_METHOD

METHOD PUBLIC TestGetSerializedDataLengthWithEmptyObject
VAR
	jsonSerializer : JsonSerializer;
	rawObject : STRING := '{}';
	length : UDINT;
	expected : UDINT := 3;
END_VAR
TEST('TestGetSerializedDataLengthWithEmptyObject');

jsonSerializer.AddRawJson(rawObject);
length := jsonSerializer.GetSerializedDataLength();

AssertEquals(
	Expected := expected,
	Actual := length,
	Message := 'Did not produce the expected JSON string length'
);

TEST_FINISHED();
END_METHOD

METHOD PUBLIC TestGetSerializedDataLengthWithSimpleObject
VAR
	jsonSerializer : JsonSerializer;
	rawObject : STRING := '{"foo":"bar"}';
	length : UDINT;
	expected : UDINT := 14;
END_VAR
TEST('TestGetSerializedDataLength');

jsonSerializer.AddRawJson(rawObject);
length := jsonSerializer.GetSerializedDataLength();

AssertEquals(
	Expected := expected,
	Actual := length,
	Message := 'Did not produce the expected JSON string length'
);

TEST_FINISHED();
END_METHOD

METHOD PUBLIC TestReset
VAR
	jsonSerializer : JsonSerializer;
	rawObject : STRING := '{"foo":"bar"}';
	out : STRING;
	expected : STRING := '';
END_VAR
TEST('TestReset');

jsonSerializer.AddRawJson(rawObject);
jsonSerializer.Reset();
jsonSerializer.TryGetSerializedData(ADR(out),SIZEOF(out));

AssertEquals(
	Expected := expected,
	Actual := out,
	Message := 'Did not reset'
);

TEST_FINISHED();
END_METHOD

METHOD PUBLIC TestSerializeArray
VAR
	jsonSerializer : JsonSerializer;
	out : STRING;
	expected : STRING := '[123,true,"foobar",null]';
END_VAR
TEST('TestSerializeArray');

jsonSerializer.StartArray();
jsonSerializer.AddDint(123);
jsonSerializer.AddBool(TRUE);
jsonSerializer.AddString('foobar');
jsonSerializer.AddNull();
jsonSerializer.EndArray();

jsonSerializer.TryGetSerializedData(ADR(out),SIZEOF(out));

AssertEquals(
	Expected := expected,
	Actual := out,
	Message := 'Did not produce the expected JSON string for the array'
);

TEST_FINISHED();
END_METHOD

METHOD PUBLIC TestSerializeObject
VAR
	jsonSerializer : JsonSerializer;
	out : STRING;
	expected : STRING := '{"dint":123,"bool":true,"string":"foobar","null":null}';
END_VAR
TEST('TestSerializeObject');

jsonSerializer.StartObject();
jsonSerializer.AddKeyDint('dint',123);
jsonSerializer.AddKeyBool('bool',TRUE);
jsonSerializer.AddKeyString('string','foobar');
jsonSerializer.AddKeyNull('null');
jsonSerializer.EndObject();

jsonSerializer.TryGetSerializedData(ADR(out),SIZEOF(out));

AssertEquals(
	Expected := expected,
	Actual := out,
	Message := 'Did not produce the expected JSON string for the object'
);

TEST_FINISHED();
END_METHOD

END_FUNCTION_BLOCK

// ---- mobject-json/Tests/Mocks/MockSerializableUserObject.TcPOU
FUNCTION_BLOCK MockSerializableUserObject IMPLEMENTS I_Serializable
VAR
	_name : STRING;
	_age : INT;
END_VAR

PROPERTY PUBLIC Age : INT
GET
Age := _age;
END_GET
SET
_age := Age;
END_SET
END_PROPERTY

METHOD FB_init : BOOL
VAR_INPUT
	bInitRetains : BOOL; // if TRUE, the retain variables are initialized (warm start / cold start)
	bInCopyCode : BOOL;  // if TRUE, the instance afterwards gets moved into the copy code (online change)
	Name : STRING;
	Age : INT;
END_VAR
_name := Name;
_age := Age;
END_METHOD

PROPERTY PUBLIC Name : STRING
GET
Name := _name;
END_GET
SET
_name := Name;
END_SET
END_PROPERTY

METHOD SerializeWith
VAR_INPUT
	Serializer : I_Serializer;
END_VAR
Serializer.StartObject().AddKeyString('Name',_name).AddKeyInt('Age',_age).EndObject();
END_METHOD

END_FUNCTION_BLOCK

// ---- mobject-json/Tests/JsonDeserializer_TestSuite.TcPOU
FUNCTION_BLOCK JsonDeserializer_TestSuite EXTENDS TcUnit.FB_TestSuite

TestClone();
TestReset();
TestGetArray();
TestGetKeyArray();
TestGetKeyObject();
TestGetObject();
TestTryGetBase64();
TestTryGetBoolWithFalseValue();
TestTryGetBoolWithTrueValue();
TestTryGetByte();
TestTryGetHexAsBytes();
TestTryGetDateTime();
TestTryGetDcTime();
TestTryGetDint();
TestTryGetDword();
TestTryGetElement();
TestTryGetFileTime();
TestTryGetInt();
TestTryGetKeyBase64();
TestTryGetKeyBoolWithFalseBoolVariable();
TestTryGetKeyBoolWithTrueBoolVariable();
TestTryGetKeyByte();
TestTryGetKeyHexAsBytes();
TestTryGetKeyDateTime();
TestTryGetKeyDcTime();
TestTryGetKeyDint();
TestTryGetKeyDword();
TestTryGetKeyFileTime();
TestTryGetKeyInt();
TestTryGetKeyLint();
TestTryGetKeyLreal();
TestTryGetKeyLtime();
TestTryGetKeyLword();
TestTryDeserializeKeyToObject();
TestTryDeserializeKeyToObjectFailsWithMissingKey();
TestTryDeserializeKeyToObjectFailsWithInvalidKey();
TestTryGetKeyReal();
TestTryGetKeySint();
TestTryGetKeyString();
TestTryGetKeyStringEx();
TestTryGetKeyTime();
TestTryGetKeyTod();
TestTryGetKeyUdint();
TestTryGetKeyUint();
TestTryGetKeyUlint();
TestTryGetKeyUsint();
TestTryGetKeyWord();
TestTryGetLint();
TestTryGetLreal();
TestTryGetLtime();
TestTryGetLword();
TestTryDeserializeToObject();
TestTryGetReal();
TestTryGetSint();
TestTryGetString();
TestTryGetStringEx();
TestTryGetTime();
TestTryGetTod();
TestTryGetUdint();
TestTryGetUint();
TestTryGetUlint();
TestTryGetUsint();
TestTryGetWord();

METHOD PUBLIC TestClone
VAR
	jsonDeserializer : JsonDeserializer;
	clone : I_Deserializer;
    json : STRING := '{"data":100}';
    out : BYTE;
	feedback : DeserializerFeedback;
	hasDeserializer : BOOL;
    expected : BYTE := 100;
END_VAR
TEST('TestClone');

// add something to the original 
jsonDeserializer.TryLoad(json);

// deep clone
clone := jsonDeserializer.Clone();

// reset the original
jsonDeserializer.Reset();

// retreive the data from the clone
clone.TryGetKeyByte('data', out, feedback);

// clones are __NEW so must be disposed
clone.Dispose();

AssertEquals(
	Expected := expected,
	Actual := out,
	Message := 'Did not create a deep copy clone'
);

TEST_FINISHED();
END_METHOD

METHOD PUBLIC TestGetArray
VAR
    jsonDeserializer : JsonDeserializer;
	arrayDeserializer : I_Deserializer;
	elementDeserializer : I_Deserializer;
    json : STRING := '[100,200,300]';
    out : BYTE;
	feedback : DeserializerFeedback;
	hasArrayDeserializer : BOOL;
	hasElementDeserializer : BOOL;
    expected : BYTE := 100;
END_VAR
TEST('TestGetArray');

jsonDeserializer.TryLoad(json);
arrayDeserializer := jsonDeserializer.GetArray();

hasArrayDeserializer := arrayDeserializer <> 0;

IF hasArrayDeserializer THEN
	elementDeserializer := arrayDeserializer.GetElementByIndex(0);
END_IF

AssertTrue(
	Condition := hasArrayDeserializer,
	Message := 'Did not return deserializer for array'
);

hasElementDeserializer := elementDeserializer <> 0;

IF hasElementDeserializer THEN
	elementDeserializer.TryGetByte(out, feedback);
END_IF

AssertTrue(
	Condition := hasElementDeserializer,
	Message := 'Did not return deserializer for element'
);

AssertEquals(
    Expected := expected,
    Actual := out,
    Message := 'Did not produce the expected BYTE value from JSON array'
);

TEST_FINISHED();
END_METHOD

METHOD PUBLIC TestGetKeyArray
VAR
    jsonDeserializer : JsonDeserializer;
	arrayDeserializer : I_Deserializer;
	elementDeserializer : I_Deserializer;
    json : STRING := '{"myArray":[100,200,300]}';
    out : BYTE;
	feedback : DeserializerFeedback;
	hasArrayDeserializer : BOOL;
	hasElementDeserializer : BOOL;
    expected : BYTE := 100;
END_VAR
TEST('TestGetKeyArray');

jsonDeserializer.TryLoad(json);
arrayDeserializer := jsonDeserializer.GetKeyArray('myArray');

hasArrayDeserializer := arrayDeserializer <> 0;

IF hasArrayDeserializer THEN
	elementDeserializer := arrayDeserializer.GetElementByIndex(0);
END_IF

AssertTrue(
	Condition := hasArrayDeserializer,
	Message := 'Did not return deserializer for array'
);

hasElementDeserializer := elementDeserializer <> 0;

IF hasElementDeserializer THEN
	elementDeserializer.TryGetByte(out, feedback);
END_IF

AssertTrue(
	Condition := hasElementDeserializer,
	Message := 'Did not return deserializer for element'
);

AssertEquals(
    Expected := expected,
    Actual := out,
    Message := 'Did not produce the expected BYTE value from JSON array'
);

TEST_FINISHED();
END_METHOD

METHOD PUBLIC TestGetKeyObject
VAR
    jsonDeserializer : JsonDeserializer;
	objectDeserializer : I_Deserializer;
    json : STRING := '{"data":100}';
    out : BYTE;
	feedback : DeserializerFeedback;
	hasObjectDeserializer : BOOL;
    expected : BYTE := 100;
END_VAR
TEST('TestGetKeyObject');

jsonDeserializer.TryLoad(json);
objectDeserializer := jsonDeserializer.GetKeyObject('data');

hasObjectDeserializer := objectDeserializer <> 0;

IF hasObjectDeserializer THEN
	objectDeserializer.TryGetByte(out, feedback);
END_IF

AssertTrue(
	Condition := hasObjectDeserializer,
	Message := 'Did not return deserializer for object'
);

AssertEquals(
    Expected := expected,
    Actual := out,
    Message := 'Did not produce the expected BYTE value from JSON'
);

TEST_FINISHED();
END_METHOD

METHOD PUBLIC TestGetObject
VAR
    jsonDeserializer : JsonDeserializer;
	objectDeserializer : I_Deserializer;
    json : STRING := '{"data":100}';
    out : BYTE;
	feedback : DeserializerFeedback;
	hasObjectDeserializer : BOOL;
    expected : BYTE := 100;
END_VAR
TEST('TestGetObject');

jsonDeserializer.TryLoad(json);
objectDeserializer := jsonDeserializer.GetObject();

hasObjectDeserializer := objectDeserializer <> 0;

IF hasObjectDeserializer THEN
	objectDeserializer.TryGetKeyByte('data',out, feedback);
END_IF

AssertTrue(
	Condition := hasObjectDeserializer,
	Message := 'Did not return deserializer for object'
);

AssertEquals(
    Expected := expected,
    Actual := out,
    Message := 'Did not produce the expected BYTE value from JSON'
);

TEST_FINISHED();
END_METHOD

METHOD PUBLIC TestReset
VAR
	jsonDeserializer : JsonDeserializer;
    json : STRING := '100';
    out : BYTE;
	feedback : DeserializerFeedback;
    expected : BYTE := 0; 
END_VAR
TEST('TestReset');

jsonDeserializer.TryLoad(json);
jsonDeserializer.Reset();
jsonDeserializer.TryGetByte(out, feedback);

AssertEquals(
	Expected := expected,
	Actual := out,
	Message := 'Did not reset'
);

TEST_FINISHED();
END_METHOD

METHOD PUBLIC TestTryDeserializeKeyToObject
VAR
    jsonDeserializer : JsonDeserializer;
    json : STRING := '{"data":{"Name":"alice","Age":40}}';
    out : MockDeserializableUserObject;
	feedback : DeserializerFeedback;
    expectedName : STRING := 'alice';
	expectedAge : INT := 40;
	actualName : STRING;
	actualAge : INT;
END_VAR
TEST('TestTryDeserializeKeyToObject');
jsonDeserializer.TryLoad(json);
jsonDeserializer.TryDeserializeKeyToObject('data', out, feedback);

actualName := out.Name;
actualAge := out.Age;

AssertEquals(
    Expected := expectedName,
    Actual := actualName,
    Message := 'Did not produce the expected Object values from JSON'
);

AssertEquals(
    Expected := expectedAge,
    Actual := actualAge,
    Message := 'Did not produce the expected Object values from JSON'
);

TEST_FINISHED();
END_METHOD

METHOD PUBLIC TestTryDeserializeKeyToObjectFailsWithInvalidKey
VAR
    jsonDeserializer : JsonDeserializer;
    json : STRING := '{"data":{"Name":"alice","Age":40}}';
    out : MockDeserializableUserObject;
	feedback : DeserializerFeedback;
	result : BOOL;
END_VAR
TEST('TestTryDeserializeKeyToObjectFailsWithInvalidKey');
jsonDeserializer.TryLoad(json);
result := jsonDeserializer.TryDeserializeKeyToObject('', out, feedback);

AssertFalse(
	Condition := result,
	Message := 'Try returned true, even though key was invalid present');

TEST_FINISHED();
END_METHOD

METHOD PUBLIC TestTryDeserializeKeyToObjectFailsWithMissingKey
VAR
    jsonDeserializer : JsonDeserializer;
    json : STRING := '{"data":{"Name":"alice","Age":40}}';
    out : MockDeserializableUserObject;
	feedback : DeserializerFeedback;
	result : BOOL;
END_VAR
TEST('TestTryDeserializeKeyToObjectFailsWithMissingKey');
jsonDeserializer.TryLoad(json);
result := jsonDeserializer.TryDeserializeKeyToObject('test', out, feedback);

AssertFalse(
	Condition := result,
	Message := 'Try returned true, even though key was not present');

TEST_FINISHED();
END_METHOD

METHOD PUBLIC TestTryDeserializeToObject
VAR
    jsonDeserializer : JsonDeserializer;
    json : STRING := '{"Name":"alice","Age":40}';
    out : MockDeserializableUserObject;
	feedback : DeserializerFeedback;
    expectedName : STRING := 'alice';
	expectedAge : INT := 40;
	actualName : STRING;
	actualAge : INT;
END_VAR
TEST('TestTryDeserializeToObject');

jsonDeserializer.TryLoad(json);
jsonDeserializer.TryDeserializeToObject(out, feedback);

actualName := out.Name;
actualAge := out.Age;

AssertEquals(
    Expected := expectedName,
    Actual := actualName,
    Message := 'Did not produce the expected Object values from JSON'
);

AssertEquals(
    Expected := expectedAge,
    Actual := actualAge,
    Message := 'Did not produce the expected Object values from JSON'
);

TEST_FINISHED();
END_METHOD

METHOD PUBLIC TestTryGetBase64
VAR
	jsonDeserializer : JsonDeserializer;
	json : STRING := '"aGVsbG8="';
	out : ARRAY[0..4] OF BYTE;
	feedback : DeserializerFeedback;
	expected : ARRAY[0..4] OF BYTE := [104, 101, 108, 108, 111]; 
END_VAR
TEST('TestTryGetBase64');

jsonDeserializer.TryLoad(json);
jsonDeserializer.TryGetBase64(ADR(out), SIZEOF(out), feedback);

AssertEquals(
	Expected := expected,
	Actual := out,
	Message := 'Did not produce the expected Base64 encoded "hello" from JSON'
);

TEST_FINISHED();
END_METHOD

METHOD PUBLIC TestTryGetBoolWithFalseValue
VAR
	jsonDeserializer : JsonDeserializer;
	json : STRING := 'false';
	out : BOOL;
	feedback : DeserializerFeedback;
	expected : BOOL := FALSE;
END_VAR
TEST('TestTryGetBoolWithFalseValue');

jsonDeserializer.TryLoad(json);
jsonDeserializer.TryGetBool(out, feedback);

AssertEquals(
	Expected := expected,
	Actual := out,
	Message := 'Did not produce the expected JSON string for a false value'
);

TEST_FINISHED();
END_METHOD

METHOD PUBLIC TestTryGetBoolWithTrueValue
VAR
    jsonDeserializer : JsonDeserializer;
    json : STRING := 'true';
    out : BOOL;
	feedback : DeserializerFeedback;
    expected : BOOL := TRUE; 
END_VAR
TEST('TestTryGetBoolWithTrueValue');

jsonDeserializer.TryLoad(json);
jsonDeserializer.TryGetBool(out, feedback);

AssertEquals(
    Expected := expected,
    Actual := out,
    Message := 'Did not produce the expected true value from JSON'
);

TEST_FINISHED();
END_METHOD

METHOD PUBLIC TestTryGetByte
VAR
    jsonDeserializer : JsonDeserializer;
    json : STRING := '100';
    out : BYTE;
	feedback : DeserializerFeedback;
    expected : BYTE := 100; 
END_VAR
TEST('TestTryGetByte');

jsonDeserializer.TryLoad(json);
jsonDeserializer.TryGetByte(out, feedback);

AssertEquals(
    Expected := expected,
    Actual := out,
    Message := 'Did not produce the expected BYTE value from JSON'
);

TEST_FINISHED();
END_METHOD

METHOD PUBLIC TestTryGetDateTime
VAR
    jsonDeserializer : JsonDeserializer;
    json : STRING := '"2023-12-30T15:20:00"';
    out : DATE_AND_TIME;
	feedback : DeserializerFeedback;
    expected : DATE_AND_TIME := DT#2023-12-30-15:20:00; 
END_VAR
TEST('TestTryGetDateTime');

jsonDeserializer.TryLoad(json);
jsonDeserializer.TryGetDateTime(out, feedback);

AssertEquals(
    Expected := expected,
    Actual := out,
    Message := 'Did not produce the expected DATE_AND_TIME value from JSON'
);

TEST_FINISHED();
END_METHOD

METHOD PUBLIC TestTryGetDcTime
VAR
    jsonDeserializer : JsonDeserializer;
    json : STRING := '"2000-01-01T00:00:00.012345678"';
    out : DCTIME;
	feedback : DeserializerFeedback;
    expected : DCTIME := 12345678;
END_VAR
TEST('TestTryGetDcTime');

jsonDeserializer.TryLoad(json);
jsonDeserializer.TryGetDcTime(out, feedback);

AssertEquals(
    Expected := expected,
    Actual := out,
    Message := 'Did not produce the expected DCTIME value from JSON string'
);

TEST_FINISHED();
END_METHOD

METHOD PUBLIC TestTryGetDint
VAR
    jsonDeserializer : JsonDeserializer;
    json : STRING := '12345';
    out : DINT;
	feedback : DeserializerFeedback;
    expected : DINT := 12345;
END_VAR
TEST('TestTryGetDint');

jsonDeserializer.TryLoad(json);
jsonDeserializer.TryGetDint(out, feedback);

AssertEquals(
    Expected := expected,
    Actual := out,
    Message := 'Did not produce the expected DINT value from JSON'
);

TEST_FINISHED();
END_METHOD

METHOD PUBLIC TestTryGetDword
VAR
    jsonDeserializer : JsonDeserializer;
    json : STRING := '12345';
    out : DWORD;
	feedback : DeserializerFeedback;
    expected : DWORD := 12345;
END_VAR
TEST('TestTryGetDword');

jsonDeserializer.TryLoad(json);
jsonDeserializer.TryGetDword(out, feedback);

AssertEquals(
    Expected := expected,
    Actual := out,
    Message := 'Did not produce the expected DWORD value from JSON'
);

TEST_FINISHED();
END_METHOD

METHOD PUBLIC TestTryGetElement
VAR
    jsonDeserializer : JsonDeserializer;
	arrayDeserializer : I_Deserializer;
	elementDeserializer : I_Deserializer;
    json : STRING := '[100,200,300]';
    out : BYTE;
	feedback : DeserializerFeedback;
	hasArrayDeserializer : BOOL;
	hasElementDeserializer : BOOL;
    expected : BYTE := 100;
END_VAR
TEST('TestTryGetElement');

jsonDeserializer.TryLoad(json);
arrayDeserializer := jsonDeserializer.GetArray();

hasArrayDeserializer := arrayDeserializer <> 0;

IF hasArrayDeserializer THEN
	hasElementDeserializer := arrayDeserializer.TryGetElementByIndex(0, elementDeserializer, feedback);
END_IF

AssertTrue(
	Condition := hasArrayDeserializer,
	Message := 'Did not return deserializer for array'
);

IF hasElementDeserializer THEN
	elementDeserializer.TryGetByte(out, feedback);
END_IF

AssertTrue(
	Condition := hasElementDeserializer,
	Message := 'Did not return deserializer for element'
);

AssertEquals(
    Expected := expected,
    Actual := out,
    Message := 'Did not produce the expected BYTE value from JSON array'
);

TEST_FINISHED();
END_METHOD

METHOD PUBLIC TestTryGetFileTime
VAR
    jsonDeserializer : JsonDeserializer;
    json : STRING := '"1601-01-01T00:00:01.2345678"';
    out : FILETIME;
	feedback : DeserializerFeedback;
    expected : FILETIME := 12345678; 
END_VAR
TEST('TestTryGetFileTime');

jsonDeserializer.TryLoad(json);
jsonDeserializer.TryGetFileTime(out, feedback);

AssertEquals(
    Expected := expected,
    Actual := out,
    Message := 'Did not produce the expected FILETIME value from JSON'
);

TEST_FINISHED();
END_METHOD

METHOD PUBLIC TestTryGetHexAsBytes
VAR
    jsonDeserializer : JsonDeserializer;
    json : STRING := '"baadf00d"';
    out : ARRAY[0..3] OF BYTE;
	feedback : DeserializerFeedback;
    expected : ARRAY[0..3] OF BYTE := [16#BA, 16#AD, 16#F0, 16#0D];
END_VAR
TEST('TestTryGetHexAsBytes');

jsonDeserializer.TryLoad(json);
jsonDeserializer.TryGetHexAsBytes(ADR(out), SIZEOF(out), feedback);

AssertEquals(
    Expected := expected,
    Actual := out,
    Message := 'Did not produce the expected binary data from JSON hexadecimal string'
);

TEST_FINISHED();
END_METHOD

METHOD PUBLIC TestTryGetInt
VAR
    jsonDeserializer : JsonDeserializer;
    json : STRING := '12345';
    out : INT;
	feedback : DeserializerFeedback;
    expected : INT := 12345;
END_VAR
TEST('TestTryGetInt');

jsonDeserializer.TryLoad(json);
jsonDeserializer.TryGetInt(out, feedback);

AssertEquals(
    Expected := expected,
    Actual := out,
    Message := 'Did not produce the expected INT value from JSON'
);

TEST_FINISHED();
END_METHOD

METHOD PUBLIC TestTryGetKeyBase64
VAR
    jsonDeserializer : JsonDeserializer;
    json : STRING := '{"data":"aGVsbG8="}';
    out : ARRAY[0..4] OF BYTE;
	feedback : DeserializerFeedback;
    expected : ARRAY[0..4] OF BYTE := [104, 101, 108, 108, 111];
END_VAR
TEST('TestTryGetKeyBase64');

jsonDeserializer.TryLoad(json);
jsonDeserializer.TryGetKeyBase64('data', ADR(out), SIZEOF(out), feedback);

AssertEquals(
    Expected := expected,
    Actual := out,
    Message := 'Did not produce the expected binary data from JSON Base64 encoded "hello"'
);

TEST_FINISHED();
END_METHOD

METHOD PUBLIC TestTryGetKeyBoolWithFalseBoolVariable
VAR
    jsonDeserializer : JsonDeserializer;
    json : STRING := '{"data":false}';
    out : BOOL;
	feedback : DeserializerFeedback;
    expected : BOOL := FALSE;
END_VAR
TEST('TestTryGetKeyBoolWithFalseBoolVariable');

jsonDeserializer.TryLoad(json);
jsonDeserializer.TryGetKeyBool('data', out, feedback);

AssertEquals(
    Expected := expected,
    Actual := out,
    Message := 'Did not produce the expected boolean value from JSON for a false value'
);

TEST_FINISHED();
END_METHOD

METHOD PUBLIC TestTryGetKeyBoolWithTrueBoolVariable
VAR
    jsonDeserializer : JsonDeserializer;
    json : STRING := '{"data":true}';
    out : BOOL;
	feedback : DeserializerFeedback;
    expected : BOOL := TRUE;
END_VAR
TEST('TestTryGetKeyBoolWithTrueBoolVariable');

jsonDeserializer.TryLoad(json);
jsonDeserializer.TryGetKeyBool('data', out, feedback);

AssertEquals(
    Expected := expected,
    Actual := out,
    Message := 'Did not produce the expected boolean value from JSON for a true value'
);

TEST_FINISHED();
END_METHOD

METHOD PUBLIC TestTryGetKeyByte
VAR
    jsonDeserializer : JsonDeserializer;
    json : STRING := '{"data":100}';
    out : BYTE;
	feedback : DeserializerFeedback;
    expected : BYTE := 100;
END_VAR
TEST('TestTryGetKeyByte');

jsonDeserializer.TryLoad(json);
jsonDeserializer.TryGetKeyByte('data', out, feedback);

AssertEquals(
    Expected := expected,
    Actual := out,
    Message := 'Did not produce the expected BYTE value from JSON'
);

TEST_FINISHED();
END_METHOD

METHOD PUBLIC TestTryGetKeyDateTime
VAR
    jsonDeserializer : JsonDeserializer;
    json : STRING := '{"data":"2023-12-30T15:20:00"}';
    out : DATE_AND_TIME;
	feedback : DeserializerFeedback;
    expected : DATE_AND_TIME := DT#2023-12-30-15:20:00;
END_VAR
TEST('TestTryGetKeyDateTime');

jsonDeserializer.TryLoad(json);
jsonDeserializer.TryGetKeyDateTime('data', out, feedback);

AssertEquals(
    Expected := expected,
    Actual := out,
    Message := 'Did not produce the expected DATE_AND_TIME value from JSON'
);

TEST_FINISHED();
END_METHOD

METHOD PUBLIC TestTryGetKeyDcTime
VAR
    jsonDeserializer : JsonDeserializer;
    json : STRING := '{"data":"2000-01-01T00:00:00.012345678"}';
    out : DCTIME;
	feedback : DeserializerFeedback;
    expected : DCTIME := 12345678;
END_VAR
TEST('TestTryGetKeyDcTime');

jsonDeserializer.TryLoad(json);
jsonDeserializer.TryGetKeyDcTime('data', out, feedback);

AssertEquals(
    Expected := expected,
    Actual := out,
    Message := 'Did not produce the expected DCTIME value from JSON string'
);

TEST_FINISHED();
END_METHOD

METHOD PUBLIC TestTryGetKeyDint
VAR
    jsonDeserializer : JsonDeserializer;
    json : STRING := '{"data":12345}';
    out : DINT;
	feedback : DeserializerFeedback;
    expected : DINT := 12345;
END_VAR
TEST('TestTryGetKeyDint');

jsonDeserializer.TryLoad(json);
jsonDeserializer.TryGetKeyDint('data', out, feedback);

AssertEquals(
    Expected := expected,
    Actual := out,
    Message := 'Did not produce the expected DINT value from JSON'
);

TEST_FINISHED();
END_METHOD

METHOD PUBLIC TestTryGetKeyDword
VAR
    jsonDeserializer : JsonDeserializer;
    json : STRING := '{"data":12345}';
    out : DWORD;
	feedback : DeserializerFeedback;
    expected : DWORD := 12345;
END_VAR
TEST('TestTryGetKeyDword');

jsonDeserializer.TryLoad(json);
jsonDeserializer.TryGetKeyDword('data', out, feedback);

AssertEquals(
    Expected := expected,
    Actual := out,
    Message := 'Did not produce the expected DWORD value from JSON'
);

TEST_FINISHED();
END_METHOD

METHOD PUBLIC TestTryGetKeyFileTime
VAR
    jsonDeserializer : JsonDeserializer;
    json : STRING := '{"data":"1601-01-01T00:00:01.2345678"}';
    out : FILETIME;
	feedback : DeserializerFeedback;
    expected : FILETIME := 12345678;
END_VAR
TEST('TestTryGetKeyFileTime');

jsonDeserializer.TryLoad(json);
jsonDeserializer.TryGetKeyFileTime('data', out, feedback);

AssertEquals(
    Expected := expected,
    Actual := out,
    Message := 'Did not produce the expected FILETIME value from JSON string'
);

TEST_FINISHED();
END_METHOD

METHOD PUBLIC TestTryGetKeyHexAsBytes
VAR
    jsonDeserializer : JsonDeserializer;
    json : STRING := '{"data":"baadf00d"}';
    out : ARRAY[0..3] OF BYTE;
	feedback : DeserializerFeedback;
    expected : ARRAY[0..3] OF BYTE := [16#BA, 16#AD, 16#F0, 16#0D];
END_VAR
TEST('TestTryGetKeyHexAsBytes');

jsonDeserializer.TryLoad(json);
jsonDeserializer.TryGetKeyHexAsBytes('data', ADR(out), SIZEOF(out), feedback);

AssertEquals(
    Expected := expected,
    Actual := out,
    Message := 'Did not produce the expected binary data from JSON hexadecimal string'
);

TEST_FINISHED();
END_METHOD

METHOD PUBLIC TestTryGetKeyInt
VAR
    jsonDeserializer : JsonDeserializer;
    json : STRING := '{"data":12345}';
    out : INT;
	feedback : DeserializerFeedback;
    expected : INT := 12345;
END_VAR
TEST('TestTryGetKeyInt');

jsonDeserializer.TryLoad(json);
jsonDeserializer.TryGetKeyInt('data', out, feedback);

AssertEquals(
    Expected := expected,
    Actual := out,
    Message := 'Did not produce the expected INT value from JSON'
);

TEST_FINISHED();
END_METHOD

METHOD PUBLIC TestTryGetKeyLint
VAR
    jsonDeserializer : JsonDeserializer;
    json : STRING := '{"data":9223372036854775807}';
    out : LINT;
	feedback : DeserializerFeedback;
    expected : LINT := 9223372036854775807;
END_VAR
TEST('TestTryGetKeyLint');

jsonDeserializer.TryLoad(json);
jsonDeserializer.TryGetKeyLint('data', out, feedback);

AssertEquals(
    Expected := expected,
    Actual := out,
    Message := 'Did not produce the expected LINT value from JSON'
);

TEST_FINISHED();
END_METHOD

METHOD PUBLIC TestTryGetKeyLreal
VAR
    jsonDeserializer : JsonDeserializer;
    json : STRING := '{"data":123456.789}';
    out : LREAL;
	feedback : DeserializerFeedback;
    expected : LREAL := 123456.789;
END_VAR
TEST('TestTryGetKeyLreal');

jsonDeserializer.TryLoad(json);
jsonDeserializer.TryGetKeyLreal('data', out, feedback);

AssertEquals(
    Expected := expected,
    Actual := out,
    Message := 'Did not produce the expected LREAL value from JSON'
);

TEST_FINISHED();
END_METHOD

METHOD PUBLIC TestTryGetKeyLtime
VAR
    jsonDeserializer : JsonDeserializer;
    json : STRING := '{"data":"LTIME#100d2h30m40s500ms600us700ns"}';
    out : LTIME;
	feedback : DeserializerFeedback;
    expected : LTIME := LTIME#100D2H30M40S500MS600US700NS;
END_VAR
TEST('TestTryGetKeyLtime');

jsonDeserializer.TryLoad(json);
jsonDeserializer.TryGetKeyLtime('data', out, feedback);

AssertEquals(
    Expected := expected,
    Actual := out,
    Message := 'Did not produce the expected LTIME value from JSON string'
);

TEST_FINISHED();
END_METHOD

METHOD PUBLIC TestTryGetKeyLword
VAR
    jsonDeserializer : JsonDeserializer;
    json : STRING := '{"data":9223372036854775807}';
    out : LWORD;
	feedback : DeserializerFeedback;
    expected : LWORD := 9223372036854775807;
END_VAR
TEST('TestTryGetKeyLword');

jsonDeserializer.TryLoad(json);
jsonDeserializer.TryGetKeyLword('data', out, feedback);

AssertEquals(
    Expected := expected,
    Actual := out,
    Message := 'Did not produce the expected LWORD value from JSON'
);

TEST_FINISHED();
END_METHOD

METHOD PUBLIC TestTryGetKeyReal
VAR
    jsonDeserializer : JsonDeserializer;
    json : STRING := '{"data":123.4}';
    out : REAL;
	feedback : DeserializerFeedback;
    expected : REAL := 123.4;
END_VAR
TEST('TestTryGetKeyReal');

jsonDeserializer.TryLoad(json);
jsonDeserializer.TryGetKeyReal('data', out, feedback);

AssertEquals(
    Expected := expected,
    Actual := out,
    Message := 'Did not produce the expected REAL value from JSON'
);

TEST_FINISHED();
END_METHOD

METHOD PUBLIC TestTryGetKeySint
VAR
    jsonDeserializer : JsonDeserializer;
    json : STRING := '{"data":123}';
    out : SINT;
	feedback : DeserializerFeedback;
    expected : SINT := 123;
END_VAR
TEST('TestTryGetKeySint');

jsonDeserializer.TryLoad(json);
jsonDeserializer.TryGetKeySint('data', out, feedback);

AssertEquals(
    Expected := expected,
    Actual := out,
    Message := 'Did not produce the expected SINT value from JSON'
);

TEST_FINISHED();
END_METHOD

METHOD PUBLIC TestTryGetKeyString
VAR
    jsonDeserializer : JsonDeserializer;
    json : T_MAXSTRING := '{"data":"foobar"}';
    out : T_MAXSTRING;
	feedback : DeserializerFeedback;
    expected : T_MAXSTRING := 'foobar';
END_VAR
TEST('TestTryGetKeyString');

jsonDeserializer.TryLoad(json);
jsonDeserializer.TryGetKeyString('data', out, feedback);

AssertEquals(
    Expected := expected,
    Actual := out,
    Message := 'Did not produce the expected STRING value from JSON'
);

TEST_FINISHED();
END_METHOD

METHOD PUBLIC TestTryGetKeyStringEx
VAR
    jsonDeserializer : JsonDeserializer;
    json : T_MAXSTRING := '{"data":"---------|---------|---------|---------|---------|---------|---------|---------|---------|"}';
    out : T_MAXSTRING;
	feedback : DeserializerFeedback;
    expected : T_MAXSTRING := '---------|---------|---------|---------|---------|---------|---------|---------|---------|'; // 90 characters
END_VAR
TEST('TestTryGetKeyStringEx');

jsonDeserializer.TryLoad(json);
jsonDeserializer.TryGetKeyStringEx('data', ADR(out), SIZEOF(out), feedback);

AssertEquals(
    Expected := expected,
    Actual := out,
    Message := 'Did not produce the expected STRING value from JSON'
);

TEST_FINISHED();
END_METHOD

METHOD PUBLIC TestTryGetKeyTime
VAR
    jsonDeserializer : JsonDeserializer;
    json : STRING := '{"data":"T#49d17h2m47s295ms"}';
    out : TIME;
	feedback : DeserializerFeedback;
    expected : TIME := T#49D17H2M47S295MS;
END_VAR
TEST('TestTryGetKeyTime');

jsonDeserializer.TryLoad(json);
jsonDeserializer.TryGetKeyTime('data', out, feedback);

AssertEquals(
    Expected := expected,
    Actual := out,
    Message := 'Did not produce the expected TIME value from JSON'
);

TEST_FINISHED();
END_METHOD

METHOD PUBLIC TestTryGetKeyTod
VAR
    jsonDeserializer : JsonDeserializer;
    json : STRING := '{"data":"TOD#23:01:23.456"}';
    out : TOD;
	feedback : DeserializerFeedback;
    expected : TOD := TOD#23:01:23.456;
END_VAR
TEST('TestTryGetKeyTod');

jsonDeserializer.TryLoad(json);
jsonDeserializer.TryGetKeyTod('data', out, feedback);

AssertEquals(
    Expected := expected,
    Actual := out,
    Message := 'Did not produce the expected TOD value from JSON'
);

TEST_FINISHED();
END_METHOD

METHOD PUBLIC TestTryGetKeyUdint
VAR
    jsonDeserializer : JsonDeserializer;
    json : STRING := '{"data":123456}';
    out : UDINT;
	feedback : DeserializerFeedback;
    expected : UDINT := 123456;
END_VAR
TEST('TestTryGetKeyUdint');

jsonDeserializer.TryLoad(json);
jsonDeserializer.TryGetKeyUdint('data', out, feedback);

AssertEquals(
    Expected := expected,
    Actual := out,
    Message := 'Did not produce the expected UDINT value from JSON'
);

TEST_FINISHED();
END_METHOD

METHOD PUBLIC TestTryGetKeyUint
VAR
    jsonDeserializer : JsonDeserializer;
    json : STRING := '{"data":12345}';
    out : UINT;
	feedback : DeserializerFeedback;
    expected : UINT := 12345;
END_VAR
TEST('TestTryGetKeyUint');

jsonDeserializer.TryLoad(json);
jsonDeserializer.TryGetKeyUint('data', out, feedback);

AssertEquals(
    Expected := expected,
    Actual := out,
    Message := 'Did not produce the expected UINT value from JSON'
);

TEST_FINISHED();
END_METHOD

METHOD PUBLIC TestTryGetKeyUlint
VAR
    jsonDeserializer : JsonDeserializer;
    json : STRING := '{"data":9223372036854775807}';
    out : ULINT;
	feedback : DeserializerFeedback;
    expected : ULINT := 9223372036854775807;
END_VAR
TEST('TestTryGetKeyUlint');

jsonDeserializer.TryLoad(json);
jsonDeserializer.TryGetKeyUlint('data', out, feedback);

AssertEquals(
    Expected := expected,
    Actual := out,
    Message := 'Did not produce the expected ULINT value from JSON'
);

TEST_FINISHED();
END_METHOD

METHOD PUBLIC TestTryGetKeyUsint
VAR
    jsonDeserializer : JsonDeserializer;
    json : STRING := '{"data":123}';
    out : USINT;
	feedback : DeserializerFeedback;
    expected : USINT := 123;
END_VAR
TEST('TestTryGetKeyUsint');

jsonDeserializer.TryLoad(json);
jsonDeserializer.TryGetKeyUsint('data', out, feedback);

AssertEquals(
    Expected := expected,
    Actual := out,
    Message := 'Did not produce the expected USINT value from JSON'
);

TEST_FINISHED();
END_METHOD

METHOD PUBLIC TestTryGetKeyWord
VAR
    jsonDeserializer : JsonDeserializer;
    json : STRING := '{"data":12345}';
    out : WORD;
	feedback : DeserializerFeedback;
    expected : WORD := 12345;
END_VAR
TEST('TestTryGetKeyWord');

jsonDeserializer.TryLoad(json);
jsonDeserializer.TryGetKeyWord('data', out, feedback);

AssertEquals(
    Expected := expected,
    Actual := out,
    Message := 'Did not produce the expected WORD value from JSON'
);

TEST_FINISHED();
END_METHOD

METHOD PUBLIC TestTryGetLint
VAR
    jsonDeserializer : JsonDeserializer;
    json : STRING := '9223372036854775807';
    out : LINT;
	feedback : DeserializerFeedback;
    expected : LINT := 9223372036854775807;
END_VAR
TEST('TestTryGetLint');

jsonDeserializer.TryLoad(json);
jsonDeserializer.TryGetLint(out, feedback);

AssertEquals(
    Expected := expected,
    Actual := out,
    Message := 'Did not produce the expected LINT value from JSON'
);

TEST_FINISHED();
END_METHOD

METHOD PUBLIC TestTryGetLreal
VAR
    jsonDeserializer : JsonDeserializer;
    json : STRING := '123456.789';
    out : LREAL;
	feedback : DeserializerFeedback;
    expected : LREAL := 123456.789;
END_VAR
TEST('TestTryGetLreal');

jsonDeserializer.TryLoad(json);
jsonDeserializer.TryGetLreal(out, feedback);

AssertEquals(
    Expected := expected,
    Actual := out,
    Message := 'Did not produce the expected LREAL value from JSON'
);

TEST_FINISHED();
END_METHOD

METHOD PUBLIC TestTryGetLtime
VAR
    jsonDeserializer : JsonDeserializer;
    json : STRING := '"LTIME#100d2h30m40s500ms600us700ns"';
    out : LTIME;
	feedback : DeserializerFeedback;
    expected : LTIME := LTIME#100D2H30M40S500MS600US700NS;
END_VAR
TEST('TestTryGetLtime');

jsonDeserializer.TryLoad(json);
jsonDeserializer.TryGetLtime(out, feedback);

AssertEquals(
    Expected := expected,
    Actual := out,
    Message := 'Did not produce the expected LTIME value from JSON string'
);

TEST_FINISHED();
END_METHOD

METHOD PUBLIC TestTryGetLword
VAR
    jsonDeserializer : JsonDeserializer;
    json : STRING := '9223372036854775807';
    out : LWORD;
	feedback : DeserializerFeedback;
    expected : LWORD := 9223372036854775807;
END_VAR
TEST('TestTryGetLword');

jsonDeserializer.TryLoad(json);
jsonDeserializer.TryGetLword(out, feedback);

AssertEquals(
    Expected := expected,
    Actual := out,
    Message := 'Did not produce the expected LWORD value from JSON'
);

TEST_FINISHED();
END_METHOD

METHOD PUBLIC TestTryGetReal
VAR
    jsonDeserializer : JsonDeserializer;
    json : STRING := '123.4';
    out : REAL;
	feedback : DeserializerFeedback;
    expected : REAL := 123.4;
END_VAR
TEST('TestTryGetReal');

jsonDeserializer.TryLoad(json);
jsonDeserializer.TryGetReal(out, feedback);

AssertEquals(
    Expected := expected,
    Actual := out,
    Message := 'Did not produce the expected REAL value from JSON'
);

TEST_FINISHED();
END_METHOD

METHOD PUBLIC TestTryGetSint
VAR
    jsonDeserializer : JsonDeserializer;
    json : STRING := '123';
    out : SINT;
	feedback : DeserializerFeedback;
    expected : SINT := 123;
END_VAR
TEST('TestTryGetSint');

jsonDeserializer.TryLoad(json);
jsonDeserializer.TryGetSint(out, feedback);

AssertEquals(
    Expected := expected,
    Actual := out,
    Message := 'Did not produce the expected SINT value from JSON'
);

TEST_FINISHED();
END_METHOD

METHOD PUBLIC TestTryGetString
VAR
    jsonDeserializer : JsonDeserializer;
    json : T_MAXSTRING := '"foobar"';
    out : T_MAXSTRING;
	feedback : DeserializerFeedback;
    expected : T_MAXSTRING := 'foobar';
END_VAR
TEST('TestTryGetString');

jsonDeserializer.TryLoad(json);
jsonDeserializer.TryGetString(out, feedback);

AssertEquals(
    Expected := expected,
    Actual := out,
    Message := 'Did not produce the expected STRING value from JSON'
);

TEST_FINISHED();
END_METHOD

METHOD PUBLIC TestTryGetStringEx
VAR
    jsonDeserializer : JsonDeserializer;
    json : T_MAXSTRING := '"---------|---------|---------|---------|---------|---------|---------|---------|---------|"';
    out : T_MAXSTRING;
	feedback : DeserializerFeedback;
    expected : T_MAXSTRING := '---------|---------|---------|---------|---------|---------|---------|---------|---------|'; // 90 characters
END_VAR
TEST('TestTryGetStringEx');

jsonDeserializer.TryLoad(json);
jsonDeserializer.TryGetStringEx(Adr(out), sizeof(out), feedback);

AssertEquals(
    Expected := expected,
    Actual := out,
    Message := 'Did not produce the expected STRING value from JSON'
);

TEST_FINISHED();
END_METHOD

METHOD PUBLIC TestTryGetTime
VAR
    jsonDeserializer : JsonDeserializer;
    json : STRING := '"T#49d17h2m47s295ms"';
    out : TIME;
	feedback : DeserializerFeedback;
    expected : TIME := T#49D17H2M47S295MS;
END_VAR
TEST('TestTryGetTime');

jsonDeserializer.TryLoad(json);
jsonDeserializer.TryGetTime(out, feedback);

AssertEquals(
    Expected := expected,
    Actual := out,
    Message := 'Did not produce the expected TIME value from JSON'
);

TEST_FINISHED();
END_METHOD

METHOD PUBLIC TestTryGetTod
VAR
    jsonDeserializer : JsonDeserializer;
    json : STRING := '"TOD#23:01:23.456"';
    out : TOD;
	feedback : DeserializerFeedback;
    expected : TOD := TOD#23:01:23.456;
END_VAR
TEST('TestTryGetTod');

jsonDeserializer.TryLoad(json);
jsonDeserializer.TryGetTod(out, feedback);

AssertEquals(
    Expected := expected,
    Actual := out,
    Message := 'Did not produce the expected TOD value from JSON string'
);

TEST_FINISHED();
END_METHOD

METHOD PUBLIC TestTryGetUdint
VAR
    jsonDeserializer : JsonDeserializer;
    json : STRING := '123456';
    out : UDINT;
	feedback : DeserializerFeedback;
    expected : UDINT := 123456;
END_VAR
TEST('TestTryGetUdint');

jsonDeserializer.TryLoad(json);
jsonDeserializer.TryGetUdint(out, feedback);

AssertEquals(
    Expected := expected,
    Actual := out,
    Message := 'Did not produce the expected UDINT value from JSON'
);

TEST_FINISHED();
END_METHOD

METHOD PUBLIC TestTryGetUint
VAR
    jsonDeserializer : JsonDeserializer;
    json : STRING := '12345';
    out : UINT;
	feedback : DeserializerFeedback;
    expected : UINT := 12345;
END_VAR
TEST('TestTryGetUint');

jsonDeserializer.TryLoad(json);
jsonDeserializer.TryGetUint(out, feedback);

AssertEquals(
    Expected := expected,
    Actual := out,
    Message := 'Did not produce the expected UINT value from JSON'
);

TEST_FINISHED();
END_METHOD

METHOD PUBLIC TestTryGetUlint
VAR
    jsonDeserializer : JsonDeserializer;
    json : STRING := '9223372036854775807';
    out : ULINT;
	feedback : DeserializerFeedback;
    expected : ULINT := 9223372036854775807;
END_VAR
TEST('TestTryGetUlint');

jsonDeserializer.TryLoad(json);
jsonDeserializer.TryGetUlint(out, feedback);

AssertEquals(
    Expected := expected,
    Actual := out,
    Message := 'Did not produce the expected ULINT value from JSON'
);

TEST_FINISHED();
END_METHOD

METHOD PUBLIC TestTryGetUsint
VAR
    jsonDeserializer : JsonDeserializer;
    json : STRING := '123';
    out : USINT;
	feedback : DeserializerFeedback;
    expected : USINT := 123;
END_VAR
TEST('TestTryGetUsint');

jsonDeserializer.TryLoad(json);
jsonDeserializer.TryGetUsint(out, feedback);

AssertEquals(
    Expected := expected,
    Actual := out,
    Message := 'Did not produce the expected USINT value from JSON'
);

TEST_FINISHED();
END_METHOD

METHOD PUBLIC TestTryGetWord
VAR
    jsonDeserializer : JsonDeserializer;
    json : STRING := '12345';
    out : WORD;
	feedback : DeserializerFeedback;
    expected : WORD := 12345;
END_VAR
TEST('TestTryGetWord');

jsonDeserializer.TryLoad(json);
jsonDeserializer.TryGetWord(out, feedback);

AssertEquals(
    Expected := expected,
    Actual := out,
    Message := 'Did not produce the expected WORD value from JSON "12345"'
);

TEST_FINISHED();
END_METHOD

END_FUNCTION_BLOCK

// ---- mobject-json/Tests/Mocks/MockDeserializableUserObject.TcPOU
FUNCTION_BLOCK MockDeserializableUserObject IMPLEMENTS I_Deserializable
VAR
	_name : T_MAXSTRING;
	_age : INT;
END_VAR

PROPERTY PUBLIC Age : INT
GET
Age := _age;
END_GET
SET
_age := Age;
END_SET
END_PROPERTY

METHOD PRIVATE CreateMissingKeyError : I_Error
VAR_INPUT
END_VAR
END_METHOD

PROPERTY PUBLIC Name : T_MAXSTRING
GET
Name := _name;
END_GET
SET
_name := Name;
END_SET
END_PROPERTY

METHOD TryDeserializeFrom : BOOL
VAR_INPUT
	Deserializer : I_Deserializer;
	Feedback : I_DeserializerFeedback;
END_VAR
IF NOT Deserializer.TryGetKeyString('Name',_name, Feedback) THEN
	RETURN;
END_IF

IF NOT Deserializer.TryGetKeyInt('Age',_age, Feedback) THEN
	RETURN;
END_IF

TryDeserializeFrom := TRUE;
END_METHOD

END_FUNCTION_BLOCK

// ---- mobject-json/Tests/JsonDeserializerArrayForwardEnumerator_TestSuite.TcPOU
FUNCTION_BLOCK JsonDeserializerArrayForwardEnumerator_TestSuite EXTENDS TcUnit.FB_TestSuite
VAR
END_VAR

TestIsValidAtStart();
TestIsNotValidAfterParentReset();
TestMoveNextReturnsFalseAtTheEnd();
TestMoveNextReturnsTrueSingleItem();
TestMoveNextReturnsFalseWhenEmpty();
TestMoveNextReturnsTrueMultipleItems();
TestEnumerateThroughArrayOfInts();
TestEnumerateThroughArrayOfStrings();
TestEnumerateThroughArrayOfObjects();

METHOD PRIVATE TestEnumerateThroughArrayOfInts
VAR
	jsonDeserializer : JsonDeserializer;
	enumerator : I_DeserializerArrayForwardEnumerator;
    json : STRING := '[1, 2, 3]';
	out1, out2, out3 : INT;
	feedback1, feedback2, feedback3 : DeserializerFeedback;
	expected1 : INT := 1;
	expected2 : INT := 2;
	expected3 : INT := 3;
	result : BOOL;
END_VAR
TEST('TestEnumerateThroughArrayOfInts');

jsonDeserializer.TryLoad(json);
enumerator := jsonDeserializer.GetArrayEnumerator();

enumerator.MoveNext();
enumerator.Current.TryGetInt(out1, feedback1);

enumerator.MoveNext();
enumerator.Current.TryGetInt(out2, feedback2);

enumerator.MoveNext();
enumerator.Current.TryGetInt(out3, feedback3);

enumerator.Dispose();

AssertEquals(
	Expected := expected1,
	Actual := out1,
	Message := 'Did not produce the expected result'
);

AssertEquals(
	Expected := expected2,
	Actual := out2,
	Message := 'Did not produce the expected result'
);

AssertEquals(
	Expected := expected3,
	Actual := out3,
	Message := 'Did not produce the expected result'
);
	
TEST_FINISHED();
END_METHOD

METHOD PRIVATE TestEnumerateThroughArrayOfObjects
VAR
	jsonDeserializer : JsonDeserializer;
	enumerator : I_DeserializerArrayForwardEnumerator;
    json : T_MAXSTRING := '[{"name":"hello"}, {"name":"world"}, {"name":"foobar"}]';
	out1, out2, out3 : T_MAXSTRING;
	feedback1, feedback2, feedback3 : DeserializerFeedback;
	expected1 : T_MAXSTRING := 'hello';
	expected2 : T_MAXSTRING := 'world';
	expected3 : T_MAXSTRING := 'foobar';
	result : BOOL;
END_VAR
TEST('TestEnumerateThroughArrayOfObjects');

jsonDeserializer.TryLoad(json);
enumerator := jsonDeserializer.GetArrayEnumerator();

enumerator.MoveNext();
enumerator.Current.TryGetKeyString('name', out1, feedback1);

enumerator.MoveNext();
enumerator.Current.TryGetKeyString('name', out2, feedback2);

enumerator.MoveNext();
enumerator.Current.TryGetKeyString('name', out3, feedback3);

enumerator.Dispose();

AssertEquals(
	Expected := expected1,
	Actual := out1,
	Message := 'Did not produce the expected result'
);

AssertEquals(
	Expected := expected2,
	Actual := out2,
	Message := 'Did not produce the expected result'
);

AssertEquals(
	Expected := expected3,
	Actual := out3,
	Message := 'Did not produce the expected result'
);
	
TEST_FINISHED();
END_METHOD

METHOD PRIVATE TestEnumerateThroughArrayOfStrings
VAR
	jsonDeserializer : JsonDeserializer;
	enumerator : I_DeserializerArrayForwardEnumerator;
    json : T_MAXSTRING := '["one", "two", "three"]';
	out1, out2, out3 : T_MAXSTRING;
	feedback1, feedback2, feedback3 : DeserializerFeedback;
	expected1 : T_MAXSTRING := 'one';
	expected2 : T_MAXSTRING := 'two';
	expected3 : T_MAXSTRING := 'three';
	result : BOOL;
END_VAR
TEST('TestEnumerateThroughArrayOfStrings');

jsonDeserializer.TryLoad(json);
enumerator := jsonDeserializer.GetArrayEnumerator();

enumerator.MoveNext();
enumerator.Current.TryGetString(out1, feedback1);

enumerator.MoveNext();
enumerator.Current.TryGetString(out2, feedback2);

enumerator.MoveNext();
enumerator.Current.TryGetString(out3, feedback3);

enumerator.Dispose();

AssertEquals(
	Expected := expected1,
	Actual := out1,
	Message := 'Did not produce the expected result'
);

AssertEquals(
	Expected := expected2,
	Actual := out2,
	Message := 'Did not produce the expected result'
);

AssertEquals(
	Expected := expected3,
	Actual := out3,
	Message := 'Did not produce the expected result'
);
	
TEST_FINISHED();
END_METHOD

METHOD PRIVATE TestIsNotValidAfterParentReset
VAR
	jsonDeserializer : JsonDeserializer;
	enumerator : I_DeserializerArrayForwardEnumerator;
	result : BOOL;
END_VAR
TEST('TestIsNotValidAfterParentReset');

enumerator := jsonDeserializer.GetArrayEnumerator();

jsonDeserializer.Reset();
result := enumerator.IsValid;

enumerator.Dispose();

AssertFalse(
	Condition := result,
	Message := 'IsValid incorrectly returned true after parent was reset'
);

TEST_FINISHED();
END_METHOD

METHOD PRIVATE TestIsValidAtStart
VAR
	jsonDeserializer : JsonDeserializer;
	enumerator : I_DeserializerArrayForwardEnumerator;
	result : BOOL;
END_VAR
TEST('TestIsValidAtStart');

enumerator := jsonDeserializer.GetArrayEnumerator();

result := enumerator.IsValid;
enumerator.Dispose();

AssertTrue(
	Condition := result,
	Message := 'IsValid returned false'
);

TEST_FINISHED();
END_METHOD

METHOD PRIVATE TestMoveNextReturnsFalseAtTheEnd
VAR
	jsonDeserializer : JsonDeserializer;
	enumerator : I_DeserializerArrayForwardEnumerator;
    json : STRING := '[100]';
	result : BOOL;
END_VAR
TEST('CheckMoveNextReturnsFalseAtTheEnd');

jsonDeserializer.TryLoad(json);
enumerator := jsonDeserializer.GetArrayEnumerator();

enumerator.MoveNext();
result := enumerator.MoveNext();

enumerator.Dispose();

AssertFalse(result,
    'MoveNext did not correctly signal the end of the enumeration');
	
TEST_FINISHED();
END_METHOD

METHOD PRIVATE TestMoveNextReturnsFalseWhenEmpty
VAR
	jsonDeserializer : JsonDeserializer;
	enumerator : I_DeserializerArrayForwardEnumerator;
    json : STRING := '[]';
	result : BOOL;
END_VAR
TEST('CheckMoveNextReturnsFalseWhenEmpty');

jsonDeserializer.TryLoad(json);
enumerator := jsonDeserializer.GetArrayEnumerator();

result := enumerator.MoveNext();

enumerator.Dispose();

AssertFalse(result,
    'MoveNext did not correctly signal an empty array');
	
TEST_FINISHED();
END_METHOD

METHOD PRIVATE TestMoveNextReturnsTrueMultipleItems
VAR
	jsonDeserializer : JsonDeserializer;
	enumerator : I_DeserializerArrayForwardEnumerator;
    json : STRING := '[true, false, true]';
	result : BOOL;
END_VAR
TEST('CheckMoveNextReturnsTrueMultipleItems');

jsonDeserializer.TryLoad(json);
enumerator := jsonDeserializer.GetArrayEnumerator();

enumerator.MoveNext();
result := enumerator.MoveNext();

enumerator.Dispose();

AssertTrue(
	Condition := result,
	Message := 'MoveNext did not correctly signal there were more items to follow'
);
	
TEST_FINISHED();
END_METHOD

METHOD PRIVATE TestMoveNextReturnsTrueSingleItem
VAR
	jsonDeserializer : JsonDeserializer;
	enumerator : I_DeserializerArrayForwardEnumerator;
    json : STRING := '[100]';
	result : BOOL;
END_VAR
TEST('CheckMoveNextReturnsTrueSingleItem');

jsonDeserializer.TryLoad(json);
enumerator := jsonDeserializer.GetArrayEnumerator();

result := enumerator.MoveNext();

enumerator.Dispose();

AssertTrue(
	Condition := result,
	Message := 'MoveNext did not correctly signal there were more items to follow, i.e. the first item'
);
	
TEST_FINISHED();
END_METHOD

END_FUNCTION_BLOCK

// ---- mobject-server/MobjectServerUnitTests.TcPOU
PROGRAM MobjectServerUnitTests
VAR
	server_IntegrationTestSuite : Server_IntegrationTestSuite;
	chunkedRequestData_TestSuite : ChunkedRequestData_TestSuite;
	asyncResponseSessionData_TestSuite : AsyncResponseSessionData_TestSuite;
	
	initialized : BOOL;
	server : RpcServer;
	concatStringRpcHandler : ConcatStringRpcHandler;	
	syncToAsyncEchoRpcHandler : SyncToAsyncEchoRpcHandler;
	adjustableSizeReplyRpcHandler : AdjustableSizeReplyRpcHandler;
	
END_VAR

TcUnit.RUN();

// the code below is used by TwinCAT HMI implementation

IF NOT initialized THEN
	initialized := TRUE;
	server.RegisterSynchronousRpcHandler('concat',concatStringRpcHandler);
	server.RegisterSynchronousRpcHandler('asyncEcho',syncToAsyncEchoRpcHandler);
	server.RegisterSynchronousRpcHandler('adjustableSizeReply',adjustableSizeReplyRpcHandler);
END_IF

server.CyclicCall();

// this has timers inside, so must be cyclic called.
syncToAsyncEchoRpcHandler.CyclicCall();

END_PROGRAM

// ---- mobject-server/Server_IntegrationTestSuite.TcPOU
FUNCTION_BLOCK Server_IntegrationTestSuite EXTENDS TcUnit.FB_TestSuite
VAR
	// variables for TestAsyncEchoRpcCallAndResponse
	testAsyncEchoRpcCallAndResponseSetup : BOOL;
	testAsyncEchoRpcCallAndResponseServer : RpcServer;
	testAsyncEchoRpcCallAndResponseAsyncEchoRpcHandler : SyncToAsyncEchoRpcHandler;
	testAsyncEchoRpcCallAndResponseOutput : ResponseData;
	
	// variables for TestConcatRpcCallAndResponse
	testConcatRpcCallAndResponseOutput : ResponseData;
	
	// variables for TestAsyncConcatRpcCallAndResponse
	testAsyncConcatRpcCallAndResponseOutput : ResponseData;
	
	// variables for TestAsyncRejectMessage
	testAsyncRejectMessageOutput : ResponseData;
	
	// variables for TestSyncRejectMessage
	testSyncRejectMessageOutput : ResponseData;

	// variables for TestFollowupWithUnknownSessionIsRejected
	testFollowupWithUnknownSessionOutput : ResponseData;

END_VAR

TestSyncToAsyncEchoRpcCallAndResponse();
TestConcatRpcCallAndResponse();
TestConcatRpcCallAndResponseWithChunkedRequest();
TestAsyncConcatRpcCallAndResponse();
TestAsyncRejectMessage();
TestSyncRejectMessage();
TestFollowupWithUnknownSessionIsRejected();

METHOD TestAsyncConcatRpcCallAndResponse
VAR
	server : RpcServer;
	asyncConcatStringRpcHandler : AsyncConcatStringRpcHandler;
	header : T_MAXSTRING := '{"Type":"RPC 1.0","Method-Name":"concat","Content-Type":"application/json"}';
    payload : T_MAXSTRING := '{"STR1":"hello", "STR2":"world"}';
	followupHeader : T_MAXSTRING := '{"Type":"RPC 1.0","Accept":"application/json","Method-Name":"asyncEcho","Response-Id":"1","Session-Id":"1"}';
	followupPayload : T_MAXSTRING := '';
	expected : T_MAXSTRING := '"helloworld"';
	actual : T_MAXSTRING;
END_VAR
TEST('TestAsyncConcatRpcCallAndResponse');

server.RegisterAsynchronousRpcHandler('concat',asyncConcatStringRpcHandler);

testAsyncConcatRpcCallAndResponseOutput := server.HandleRequest(header,payload);
server.CyclicCall();
testAsyncConcatRpcCallAndResponseOutput := server.HandleRequest(followupHeader, followupPayload);
actual := testAsyncConcatRpcCallAndResponseOutput.Payload;

AssertEquals(
	Expected := expected, 
	Actual := actual,
	Message := 'Did not produce the expected result'
);

TEST_FINISHED();
END_METHOD

METHOD TestAsyncRejectMessage
VAR
	server : RpcServer;
	rejectWithMessageAsyncHandler : RejectWithMessageAsyncHandler;
	header : T_MAXSTRING := '{"Type":"RPC 1.0","Method-Name":"reject","Content-Type":"application/json"}';
    payload : T_MAXSTRING := '';
	followupHeader : T_MAXSTRING := '{"Response-Id":"1","Session-Id":"1"}';
	followupPayload : T_MAXSTRING := '';
	expectedFirstReply : T_MAXSTRING := '{"Session-Id":"1","Status":"Pending","Response-Id":"1","Retry-Delay":"20"}';
	expectedSecondReply : T_MAXSTRING := '{"Session-Id":"1","Status":"Error","Error-Code":"EXAMPLE_ERROR_CODE","Error-Message":"This is the reject message"}';
	actual : T_MAXSTRING;
END_VAR
TEST('TestAsyncRejectMessage');

server.RegisterAsynchronousRpcHandler('reject',rejectWithMessageAsyncHandler);

testAsyncRejectMessageOutput := server.HandleRequest(header,payload);
actual := testAsyncRejectMessageOutput.Header;

AssertEquals(
	Expected := expectedFirstReply, 
	Actual := actual,
	Message := 'Did not reply that the request was being processed'
);

server.CyclicCall();


testAsyncRejectMessageOutput := server.HandleRequest(followupHeader,followupPayload);
actual := testAsyncRejectMessageOutput.Header;


AssertEquals(
	Expected := expectedSecondReply, 
	Actual := actual,
	Message := 'Did not produce the expected result'
);

TEST_FINISHED();
END_METHOD

METHOD TestConcatRpcCallAndResponse
VAR
	server : RpcServer;
	concatStringRpcHandler : ConcatStringRpcHandler;
	header : T_MAXSTRING := '{"Type":"RPC 1.0","Method-Name":"concat","Content-Type":"application/json"}';
    payload : T_MAXSTRING := '{"STR1":"hello", "STR2":"world"}';
	expected : T_MAXSTRING := '"helloworld"';
	actual : T_MAXSTRING;
END_VAR
TEST('TestConcatRpcCallAndResponse');

server.RegisterSynchronousRpcHandler('concat',concatStringRpcHandler);

testConcatRpcCallAndResponseOutput := server.HandleRequest(header,payload);
actual := testConcatRpcCallAndResponseOutput.Payload;

AssertEquals(
	Expected := expected, 
	Actual := actual,
	Message := 'Did not produce the expected result'
);

TEST_FINISHED();
END_METHOD

METHOD TestConcatRpcCallAndResponseWithChunkedRequest
VAR
	server : RpcServer;
	concatStringRpcHandler : ConcatStringRpcHandler;
	chunk1Header : T_MAXSTRING := '{"Type":"RPC 1.0","Method-Name":"concat","Request-Id":"abc","Has-More-Chunks":true, "Chunk-Sequence":1, "Chunk-Total":2, "Content-Type":"application/json"}';
    chunk1payload : T_MAXSTRING := '{"STR1":"hello",';
	chunk2Header : T_MAXSTRING := '{"Type":"RPC 1.0","Session-Id":"1","Method-Name":"concat","Request-Id":"abc","Has-More-Chunks":false, "Chunk-Sequence":2, "Chunk-Total":2, "Content-Type":"application/json"}';
    chunk2payload : T_MAXSTRING := ' "STR2":"world"}';
	expected : T_MAXSTRING := '"helloworld"';
	out : ResponseData;
END_VAR
//TEST('TestConcatRpcCallAndResponseWithChunkedRequest');

//server.RegisterRpcHandler('concat',concatStringRpcHandler);

//out := server.HandleRequest(chunk1Header,chunk1payload);
//out := server.HandleRequest(chunk2Header,chunk2payload);

//AssertTrue(
//	Condition := expected = out.Payload,
//	Message := 'Did not produce the expected result'
//);

//TEST_FINISHED();
END_METHOD

METHOD TestFollowupWithUnknownSessionIsRejected
VAR
	server : RpcServer;
	concatStringRpcHandler : ConcatStringRpcHandler;
	// A follow-up as the client actually resends it: the original Type/Method-Name are still
	// on the header, a Response-Id has been added, and the Session-Id names a session the
	// server no longer holds (expired, or lost across a restart).
	followupHeader : T_MAXSTRING := '{"Type":"RPC 1.0","Method-Name":"concat","Content-Type":"application/json","Response-Id":"1","Session-Id":"999"}';
	followupPayload : T_MAXSTRING := '{"STR1":"hello", "STR2":"world"}';
	expectedHeader : T_MAXSTRING := '{"Status":"Error","Error-Code":"SESSION_EXPIRED","Error-Message":"The session for this follow-up has expired. The original request outcome is unknown."}';
	unexpectedPayload : T_MAXSTRING := '"helloworld"';
	actualHeader : T_MAXSTRING;
	actualPayload : T_MAXSTRING;
END_VAR
TEST('TestFollowupWithUnknownSessionIsRejected');

server.RegisterSynchronousRpcHandler('concat',concatStringRpcHandler);

testFollowupWithUnknownSessionOutput := server.HandleRequest(followupHeader,followupPayload);
actualHeader := testFollowupWithUnknownSessionOutput.Header;
actualPayload := testFollowupWithUnknownSessionOutput.Payload;

AssertEquals(
	Expected := expectedHeader,
	Actual := actualHeader,
	Message := 'A follow-up naming an unknown session should be rejected with SESSION_EXPIRED'
);

// The regression guarded against: the follow-up falling past the chunked and async
// middleware down to the rpc middleware, which still matches on Method-Name and would
// run the handler a second time.
AssertFalse(
	Condition := actualPayload = unexpectedPayload,
	Message := 'The rpc handler must not run again for a follow-up whose session has gone'
);

TEST_FINISHED();
END_METHOD

METHOD TestSyncRejectMessage
VAR
	server : RpcServer;
	rejectWithMessageSyncHandler : RejectWithMessageSyncHandler;
	header : T_MAXSTRING := '{"Type":"RPC 1.0","Method-Name":"reject","Content-Type":"application/json"}';
    payload : T_MAXSTRING := '';
	expected : T_MAXSTRING := '{"Session-Id":"1","Status":"Error","Error-Code":"EXAMPLE_ERROR_CODE","Error-Message":"This is the reject message"}';
	actual : T_MAXSTRING;
END_VAR
TEST('TestSyncRejectMessage');

server.RegisterSynchronousRpcHandler('reject',rejectWithMessageSyncHandler);

testSyncRejectMessageOutput := server.HandleRequest(header,payload);
actual := testAsyncRejectMessageOutput.Header;

AssertEquals(
	Expected := expected, 
	Actual := actual,
	Message := 'Did not produce the expected result'
);

TEST_FINISHED();
END_METHOD

METHOD TestSyncToAsyncEchoRpcCallAndResponse
VAR
	header : T_MAXSTRING := '{"Type":"RPC 1.0","Accept":"application/json","Method-Name":"asyncEcho","Content-Type":"application/json"}';
    payload : T_MAXSTRING := '{"Echo":"hello"}';
	followupHeader : T_MAXSTRING := '{"Type":"RPC 1.0","Accept":"application/json","Method-Name":"asyncEcho","Response-Id":"1","Session-Id":"1"}';
	followuPayload : T_MAXSTRING := '{"Echo":"hello"}';
	expected : T_MAXSTRING := '"hello"';
	actual : T_MAXSTRING;
END_VAR
TEST('TestAsyncEchoRpcCallAndResponse');

IF NOT testAsyncEchoRpcCallAndResponseSetup THEN
	testAsyncEchoRpcCallAndResponseServer.RegisterSynchronousRpcHandler('asyncEcho',testAsyncEchoRpcCallAndResponseAsyncEchoRpcHandler);
	testAsyncEchoRpcCallAndResponseOutput := testAsyncEchoRpcCallAndResponseServer.HandleRequest(header,payload);
	testAsyncEchoRpcCallAndResponseSetup := TRUE;	
END_IF

testAsyncEchoRpcCallAndResponseAsyncEchoRpcHandler.CyclicCall();

IF testAsyncEchoRpcCallAndResponseAsyncEchoRpcHandler.Busy THEN
	RETURN;
END_IF

testAsyncEchoRpcCallAndResponseOutput := testAsyncEchoRpcCallAndResponseServer.HandleRequest(followupHeader,followuPayload);
actual := testAsyncEchoRpcCallAndResponseOutput.Payload;

AssertEquals(
	Expected := expected, 
	Actual := actual,
	Message := 'Did not produce the expected result'
);

TEST_FINISHED();
END_METHOD

END_FUNCTION_BLOCK

// ---- mobject-server/Mocks/SyncToAsyncEchoRpcHandler.TcPOU
FUNCTION_BLOCK SyncToAsyncEchoRpcHandler IMPLEMENTS I_SynchronousRpcHandler
VAR
	asyncResponse : I_AsynchronousRpcResponse;
	result : T_MAXSTRING;
	timer : TON;
END_VAR

